C05476=1182.261,381.799,-80.874,-176.029,8.760,148.599
C05477=1182.257,382.046,-80.909,-176.028,8.763,148.599
C05478=1182.253,382.294,-80.944,-176.027,8.766,148.600
C05479=1182.249,382.541,-80.980,-176.026,8.769,148.600
C05480=1182.245,382.789,-81.014,-176.026,8.772,148.601
C05481=1182.241,383.036,-81.050,-176.024,8.776,148.601
C05482=1182.238,383.284,-81.085,-176.023,8.779,148.602
C05483=1182.233,383.531,-81.120,-176.023,8.783,148.603
C05484=1182.229,383.779,-81.155,-176.022,8.786,148.603
C05485=1182.225,384.027,-81.190,-176.021,8.789,148.604
C05486=1182.221,384.274,-81.225,-176.020,8.792,148.605
C05487=1182.217,384.521,-81.261,-176.020,8.795,148.605
C05488=1182.214,384.769,-81.296,-176.019,8.798,148.606
C05489=1182.209,385.016,-81.331,-176.019,8.800,148.606
C05490=1182.206,385.264,-81.366,-176.018,8.804,148.607
C05491=1182.202,385.512,-81.401,-176.017,8.807,148.608
C05492=1182.197,385.759,-81.436,-176.017,8.810,148.608
C05493=1182.194,386.006,-81.472,-176.016,8.813,148.609
C05494=1182.190,386.254,-81.507,-176.015,8.816,148.610
C05495=1182.185,386.501,-81.542,-176.015,8.819,148.610
C05496=1182.182,386.748,-81.577,-176.014,8.822,148.611
C05497=1182.178,386.996,-81.613,-176.013,8.825,148.611
C05498=1182.174,387.243,-81.649,-176.013,8.828,148.612
C05499=1182.170,387.491,-81.683,-176.012,8.831,148.613
C05500=1182.165,387.739,-81.719,-176.012,8.834,148.613
C05501=1182.162,387.986,-81.755,-176.012,8.837,148.614
C05502=1182.158,388.233,-81.790,-176.011,8.840,148.615
C05503=1182.154,388.481,-81.825,-176.010,8.843,148.615
C05504=1182.150,388.729,-81.860,-176.010,8.846,148.616
C05505=1182.146,388.976,-81.896,-176.009,8.849,148.616
C05506=1182.142,389.223,-81.931,-176.009,8.852,148.617
C05507=1182.138,389.470,-81.967,-176.009,8.854,148.618
C05508=1182.134,389.719,-82.001,-176.008,8.858,148.618
C05509=1182.130,389.965,-82.037,-176.008,8.860,148.619
C05510=1182.126,390.213,-82.072,-176.007,8.863,148.620
C05511=1182.122,390.461,-82.108,-176.007,8.866,148.620
C05512=1182.118,390.708,-82.144,-176.007,8.869,148.621
C05513=1182.114,390.955,-82.179,-176.007,8.871,148.622
C05514=1182.110,391.203,-82.214,-176.006,8.875,148.622
C05515=1182.106,391.451,-82.249,-176.006,8.877,148.623
C05516=1182.102,391.734,-82.290,-176.005,8.880,148.624
C05517=1182.098,392.019,-82.331,-176.005,8.884,148.624
C05518=1182.093,392.302,-82.372,-176.005,8.887,148.625
C05519=1182.088,392.586,-82.412,-176.004,8.890,148.626
C05520=1182.084,392.834,-82.448,-176.004,8.893,148.626
C05521=1182.081,393.081,-82.483,-176.004,8.895,148.627
C05522=1182.077,393.329,-82.519,-176.003,8.898,148.628
C05523=1182.072,393.576,-82.554,-176.003,8.901,148.628
C05524=1182.068,393.823,-82.590,-176.003,8.903,148.629
C05525=1182.065,394.071,-82.626,-176.003,8.907,148.630
C05526=1182.061,394.318,-82.661,-176.003,8.909,148.630
C05527=1182.057,394.565,-82.696,-176.003,8.911,148.631
C05528=1182.053,394.813,-82.732,-176.002,8.914,148.632
C05529=1182.049,395.061,-82.768,-176.002,8.917,148.632
C05530=1182.045,395.309,-82.803,-176.002,8.919,148.633
C05531=1182.041,395.556,-82.838,-176.002,8.922,148.633
C05532=1182.037,395.803,-82.874,-176.001,8.925,148.634
C05533=1182.033,396.051,-82.909,-176.001,8.928,148.635
C05534=1182.029,396.298,-82.945,-176.001,8.930,148.635
C05535=1182.025,396.546,-82.981,-176.001,8.932,148.636
C05536=1182.021,396.793,-83.016,-176.001,8.935,148.637
C05537=1182.017,397.040,-83.051,-176.001,8.937,148.637
C05538=1182.014,397.288,-83.087,-176.000,8.940,148.638
C05539=1182.009,397.535,-83.123,-176.001,8.943,148.639
C05540=1182.005,397.783,-83.159,-176.000,8.945,148.639
C05541=1182.001,398.030,-83.194,-176.000,8.948,148.640
C05542=1181.998,398.277,-83.229,-176.000,8.950,148.640
C05543=1181.993,398.525,-83.266,-176.000,8.953,148.641
C05544=1181.989,398.773,-83.301,-176.000,8.955,148.642
C05545=1181.985,399.019,-83.336,-176.000,8.957,148.642
C05546=1181.982,399.267,-83.372,-176.000,8.960,148.643
C05547=1181.977,399.515,-83.408,-176.000,8.962,148.644
C05548=1181.974,399.762,-83.444,-176.000,8.964,148.644
C05549=1181.970,400.010,-83.479,-176.000,8.967,148.645
C05550=1181.966,400.257,-83.515,-176.000,8.969,148.645
C05551=1181.961,400.504,-83.551,-176.000,8.972,148.646
C05552=1181.958,400.751,-83.587,-176.000,8.974,148.647
C05553=1181.954,400.999,-83.622,-176.000,8.977,148.647
C05554=1181.950,401.246,-83.658,-176.000,8.979,148.648
C05555=1181.946,401.494,-83.694,-176.000,8.982,148.649
C05556=1181.942,401.741,-83.729,-176.000,8.984,148.649
C05557=1181.938,401.988,-83.765,-176.000,8.986,148.650
C05558=1181.935,402.236,-83.800,-175.999,8.989,148.650
C05559=1181.930,402.484,-83.836,-176.000,8.991,148.651
C05560=1181.926,402.731,-83.872,-175.999,8.993,148.652
C05561=1181.922,402.978,-83.907,-175.999,8.996,148.652
C05562=1181.918,403.226,-83.943,-176.000,8.997,148.653
C05563=1181.914,403.473,-83.979,-176.000,9.000,148.653
C05564=1181.911,403.720,-84.015,-176.000,9.002,148.654
C05565=1181.907,403.968,-84.051,-176.000,9.005,148.654
C05566=1181.903,404.215,-84.087,-176.000,9.007,148.655
C05567=1181.898,404.462,-84.122,-175.999,9.009,148.656
C05568=1181.895,404.710,-84.157,-176.000,9.011,148.656
C05569=1181.890,404.957,-84.194,-176.000,9.013,148.657
C05570=1181.887,405.205,-84.229,-176.000,9.016,148.657
C05571=1181.883,405.452,-84.265,-176.000,9.018,148.658
C05572=1181.879,405.700,-84.302,-176.000,9.020,148.659
C05573=1181.875,405.947,-84.337,-176.000,9.022,148.659
C05574=1181.871,406.194,-84.372,-176.000,9.024,148.660
C05575=1181.867,406.441,-84.408,-176.000,9.027,148.660
C05576=1181.863,406.689,-84.444,-176.000,9.029,148.661
C05577=1181.859,406.937,-84.480,-176.000,9.031,148.662
C05578=1181.856,407.184,-84.516,-176.000,9.033,148.662
C05579=1181.852,407.431,-84.552,-176.000,9.036,148.663
C05580=1181.847,407.678,-84.587,-176.000,9.038,148.663
C05581=1181.844,407.926,-84.623,-176.000,9.039,148.664
C05582=1181.839,408.174,-84.659,-176.000,9.042,148.664
C05583=1181.836,408.420,-84.695,-176.000,9.044,148.665
C05584=1181.832,408.668,-84.731,-176.000,9.046,148.665
C05585=1181.828,408.916,-84.767,-176.001,9.048,148.666
C05586=1181.824,409.163,-84.802,-176.000,9.050,148.667
C05587=1181.820,409.410,-84.837,-176.001,9.052,148.667
C05588=1181.816,409.657,-84.874,-176.001,9.054,148.668
C05589=1181.812,409.905,-84.910,-176.000,9.057,148.668
C05590=1181.808,410.152,-84.945,-176.001,9.058,148.669
C05591=1181.804,410.400,-84.982,-176.001,9.061,148.670
C05592=1181.800,410.648,-85.017,-176.001,9.063,148.670
C05593=1181.797,410.894,-85.053,-176.001,9.064,148.671
C05594=1181.793,411.142,-85.090,-176.001,9.067,148.671
C05595=1181.788,411.389,-85.125,-176.001,9.068,148.672
C05596=1181.784,411.637,-85.161,-176.001,9.071,148.672
C05597=1181.781,411.884,-85.197,-176.001,9.073,148.673
C05598=1181.777,412.131,-85.233,-176.001,9.074,148.673
C05599=1181.773,412.379,-85.269,-176.001,9.077,148.674
C05600=1181.769,412.627,-85.304,-176.002,9.078,148.674
C05601=1181.765,412.874,-85.340,-176.001,9.081,148.675
C05602=1181.761,413.121,-85.377,-176.002,9.082,148.675
C05603=1181.757,413.368,-85.412,-176.001,9.084,148.676
C05604=1181.752,413.616,-85.448,-176.002,9.087,148.677
C05605=1181.749,413.863,-85.484,-176.002,9.088,148.677
C05606=1181.745,414.110,-85.520,-176.002,9.091,148.678
C05607=1181.741,414.358,-85.556,-176.002,9.092,148.678
C05608=1181.737,414.606,-85.592,-176.002,9.094,148.679
C05609=1181.734,414.852,-85.628,-176.002,9.096,148.679
C05610=1181.730,415.100,-85.664,-176.002,9.098,148.680
C05611=1181.726,415.348,-85.700,-176.002,9.100,148.680
C05612=1181.722,415.571,-85.732,-176.002,9.102,148.681
C05613=1181.718,415.796,-85.765,-176.002,9.103,148.681
C05614=1181.716,416.020,-85.797,-176.003,9.105,148.682
C05615=1181.714,416.244,-85.830,-176.002,9.107,148.682
C05616=1181.714,416.467,-85.862,-176.002,9.108,148.682
C05617=1181.715,416.691,-85.894,-176.003,9.110,148.683
C05618=1181.716,416.915,-85.927,-176.002,9.112,148.683
C05619=1181.719,417.138,-85.958,-176.002,9.113,148.684
C05620=1181.298,417.140,-86.000,-176.006,9.124,148.687
C05621=1181.295,416.914,-85.968,-176.005,9.123,148.687
C05622=1181.293,416.689,-85.936,-176.006,9.120,148.687
C05623=1181.293,416.464,-85.903,-176.006,9.119,148.686
C05624=1181.294,416.238,-85.871,-176.005,9.118,148.686
C05625=1181.295,416.013,-85.838,-176.006,9.115,148.685
C05626=1181.297,415.788,-85.806,-176.005,9.114,148.685
C05627=1181.301,415.563,-85.773,-176.005,9.113,148.684
C05628=1181.305,415.336,-85.740,-176.005,9.110,148.684
C05629=1181.308,415.089,-85.704,-176.005,9.109,148.683
C05630=1181.312,414.841,-85.668,-176.005,9.107,148.683
C05631=1181.316,414.594,-85.632,-176.005,9.105,148.682
C05632=1181.320,414.347,-85.596,-176.005,9.103,148.682
C05633=1181.324,414.100,-85.560,-176.005,9.101,148.681
C05634=1181.328,413.852,-85.525,-176.005,9.099,148.681
C05635=1181.332,413.605,-85.489,-176.005,9.098,148.680
C05636=1181.336,413.357,-85.452,-176.005,9.095,148.680
C05637=1181.339,413.110,-85.417,-176.005,9.094,148.679
C05638=1181.344,412.862,-85.381,-176.004,9.091,148.679
C05639=1181.347,412.615,-85.345,-176.005,9.089,148.678
C05640=1181.351,412.368,-85.309,-176.004,9.088,148.678
C05641=1181.356,412.121,-85.273,-176.005,9.085,148.677
C05642=1181.359,411.873,-85.238,-176.004,9.084,148.676
C05643=1181.364,411.625,-85.201,-176.004,9.081,148.676
C05644=1181.367,411.378,-85.165,-176.004,9.080,148.675
C05645=1181.371,411.131,-85.130,-176.004,9.078,148.675
C05646=1181.375,410.883,-85.093,-176.004,9.075,148.674
C05647=1181.379,410.636,-85.058,-176.004,9.074,148.674
C05648=1181.382,410.389,-85.022,-176.004,9.071,148.673
C05649=1181.387,410.142,-84.986,-176.004,9.069,148.672
C05650=1181.391,409.894,-84.950,-176.003,9.067,148.672
C05651=1181.395,409.647,-84.915,-176.004,9.065,148.671
C05652=1181.399,409.399,-84.878,-176.003,9.064,148.671
C05653=1181.402,409.152,-84.842,-176.003,9.061,148.670
C05654=1181.406,408.904,-84.807,-176.004,9.059,148.670
C05655=1181.410,408.657,-84.771,-176.003,9.057,148.669
C05656=1181.415,408.410,-84.735,-176.003,9.055,148.669
C05657=1181.418,408.163,-84.699,-176.003,9.053,148.668
C05658=1181.422,407.915,-84.663,-176.003,9.051,148.668
C05659=1181.426,407.668,-84.628,-176.003,9.049,148.667
C05660=1181.430,407.420,-84.592,-176.003,9.046,148.666
C05661=1181.434,407.172,-84.556,-176.003,9.044,148.666
C05662=1181.438,406.925,-84.520,-176.003,9.042,148.665
C05663=1181.442,406.679,-84.484,-176.003,9.040,148.665
C05664=1181.446,406.431,-84.448,-176.003,9.037,148.664
C05665=1181.450,406.183,-84.413,-176.002,9.036,148.664
C05666=1181.454,405.936,-84.377,-176.002,9.033,148.663
C05667=1181.458,405.688,-84.341,-176.003,9.031,148.662
C05668=1181.462,405.441,-84.305,-176.003,9.029,148.662
C05669=1181.465,405.194,-84.269,-176.003,9.026,148.661
C05670=1181.470,404.947,-84.233,-176.002,9.025,148.661
C05671=1181.474,404.699,-84.198,-176.002,9.022,148.660
C05672=1181.477,404.452,-84.162,-176.002,9.020,148.659
C05673=1181.482,404.204,-84.126,-176.002,9.017,148.659
C05674=1181.485,403.956,-84.091,-176.003,9.015,148.658
C05675=1181.489,403.709,-84.055,-176.002,9.014,148.658
C05676=1181.493,403.463,-84.019,-176.002,9.011,148.657
C05677=1181.497,403.215,-83.983,-176.002,9.009,148.656
C05678=1181.501,402.967,-83.948,-176.002,9.006,148.656
C05679=1181.505,402.720,-83.912,-176.002,9.004,148.655
C05680=1181.509,402.472,-83.876,-176.002,9.002,148.654
C05681=1181.513,402.224,-83.840,-176.003,8.999,148.654
C05682=1181.517,401.978,-83.805,-176.002,8.997,148.653
C05683=1181.521,401.730,-83.770,-176.002,8.995,148.653
C05684=1181.525,401.482,-83.733,-176.002,8.993,148.652
C05685=1181.529,401.235,-83.698,-176.002,8.990,148.651
C05686=1181.532,400.988,-83.662,-176.002,8.988,148.651
C05687=1181.537,400.740,-83.625,-176.002,8.986,148.650
C05688=1181.541,400.493,-83.590,-176.002,8.983,148.650
C05689=1181.544,400.246,-83.555,-176.002,8.981,148.649
C05690=1181.548,399.998,-83.519,-176.002,8.978,148.648
C05691=1181.553,399.751,-83.483,-176.002,8.976,148.648
C05692=1181.556,399.503,-83.447,-176.002,8.973,148.647
C05693=1181.560,399.256,-83.412,-176.002,8.971,148.647
C05694=1181.564,399.009,-83.377,-176.002,8.969,148.646
C05695=1181.569,398.761,-83.341,-176.003,8.966,148.645
C05696=1181.572,398.513,-83.305,-176.002,8.964,148.645
C05697=1181.576,398.266,-83.270,-176.003,8.961,148.644
C05698=1181.580,398.019,-83.234,-176.002,8.959,148.643
C05699=1181.585,397.771,-83.198,-176.003,8.956,148.643
C05700=1181.588,397.524,-83.163,-176.003,8.953,148.642
C05701=1181.592,397.276,-83.127,-176.003,8.951,148.642
C05702=1181.595,397.029,-83.092,-176.003,8.948,148.641
C05703=1181.600,396.782,-83.056,-176.003,8.946,148.640
C05704=1181.604,396.534,-83.020,-176.003,8.944,148.640
C05705=1181.608,396.287,-82.985,-176.004,8.941,148.639
C05706=1181.611,396.039,-82.949,-176.004,8.938,148.638
C05707=1181.616,395.792,-82.914,-176.004,8.936,148.638
C05708=1181.620,395.545,-82.878,-176.004,8.933,148.637
C05709=1181.624,395.297,-82.842,-176.004,8.930,148.636
C05710=1181.627,395.050,-82.807,-176.004,8.928,148.636
C05711=1181.631,394.802,-82.771,-176.005,8.925,148.635
C05712=1181.635,394.555,-82.736,-176.005,8.923,148.634
C05713=1181.640,394.308,-82.700,-176.005,8.920,148.634
C05714=1181.643,394.060,-82.664,-176.005,8.917,148.633
C05715=1181.647,393.813,-82.629,-176.005,8.914,148.632
C05716=1181.651,393.566,-82.594,-176.005,8.912,148.632
C05717=1181.655,393.318,-82.558,-176.006,8.909,148.631
C05718=1181.659,393.071,-82.522,-176.006,8.906,148.631
C05719=1181.663,392.822,-82.487,-176.006,8.904,148.630
C05720=1181.667,392.575,-82.451,-176.007,8.901,148.629
C05721=1181.672,392.291,-82.411,-176.007,8.898,148.629
C05722=1181.676,392.007,-82.371,-176.007,8.895,148.628
C05723=1181.680,391.723,-82.329,-176.007,8.891,148.627
C05724=1181.686,391.439,-82.289,-176.008,8.888,148.626
C05725=1181.689,391.191,-82.253,-176.008,8.886,148.626
C05726=1181.693,390.944,-82.218,-176.009,8.883,148.625
C05727=1181.697,390.697,-82.183,-176.009,8.880,148.624
C05728=1181.701,390.450,-82.147,-176.009,8.877,148.624
C05729=1181.704,390.202,-82.111,-176.009,8.874,148.623
C05730=1181.708,389.955,-82.076,-176.010,8.871,148.623
C05731=1181.713,389.707,-82.041,-176.010,8.869,148.622
C05732=1181.717,389.459,-82.005,-176.011,8.866,148.621
C05733=1181.721,389.212,-81.970,-176.012,8.863,148.621
C05734=1181.725,388.965,-81.935,-176.011,8.860,148.620
C05735=1181.729,388.718,-81.899,-176.012,8.857,148.619
C05736=1181.733,388.470,-81.864,-176.013,8.854,148.619
C05737=1181.736,388.222,-81.829,-176.013,8.851,148.618
C05738=1181.741,387.975,-81.793,-176.014,8.848,148.617
C05739=1181.744,387.728,-81.758,-176.014,8.845,148.617
C05740=1181.748,387.480,-81.722,-176.014,8.842,148.616
C05741=1181.752,387.233,-81.688,-176.015,8.839,148.616
C05742=1181.757,386.985,-81.652,-176.016,8.836,148.615
C05743=1181.761,386.737,-81.616,-176.016,8.833,148.614
C05744=1181.764,386.490,-81.581,-176.017,8.830,148.614
C05745=1181.769,386.243,-81.546,-176.017,8.827,148.613
C05746=1181.772,385.995,-81.511,-176.018,8.824,148.612
C05747=1181.776,385.748,-81.475,-176.019,8.821,148.612
C05748=1181.780,385.501,-81.440,-176.019,8.818,148.611
C05749=1181.784,385.253,-81.405,-176.020,8.815,148.610
C05750=1181.788,385.005,-81.370,-176.021,8.811,148.610
C05751=1181.792,384.758,-81.334,-176.021,8.808,148.609
C05752=1181.796,384.510,-81.300,-176.022,8.805,148.609
C05753=1181.800,384.263,-81.264,-176.023,8.802,148.608
C05754=1181.804,384.016,-81.229,-176.024,8.799,148.607
C05755=1181.808,383.768,-81.194,-176.024,8.796,148.607
C05756=1181.812,383.520,-81.158,-176.025,8.793,148.606
C05757=1181.816,383.274,-81.123,-176.026,8.790,148.606
C05758=1181.820,383.025,-81.088,-176.027,8.786,148.605
C05759=1181.824,382.778,-81.053,-176.028,8.783,148.604
C05760=1181.828,382.531,-81.018,-176.028,8.780,148.604
C05761=1181.832,382.283,-80.983,-176.029,8.777,148.603
C05762=1181.836,382.035,-80.947,-176.030,8.774,148.603
C05763=1181.840,381.788,-80.913,-176.031,8.771,148.602
C05764=1181.844,381.541,-80.877,-176.031,8.768,148.601
C05765=1181.848,381.292,-80.842,-176.033,8.764,148.601
C05766=1181.852,381.046,-80.807,-176.033,8.761,148.600
C05767=1181.856,380.798,-80.772,-176.035,8.758,148.600
C05768=1181.860,380.551,-80.737,-176.036,8.755,148.599
C05769=1181.864,380.303,-80.702,-176.036,8.752,148.599
C05770=1181.868,380.055,-80.667,-176.038,8.748,148.598
C05771=1181.872,379.808,-80.632,-176.039,8.745,148.597
C05772=1181.875,379.560,-80.597,-176.039,8.741,148.597
C05773=1181.879,379.313,-80.562,-176.040,8.738,148.596
C05774=1181.884,379.066,-80.527,-176.042,8.734,148.595
C05775=1181.887,378.818,-80.492,-176.042,8.731,148.595
C05776=1181.892,378.571,-80.457,-176.043,8.728,148.594
C05777=1181.895,378.323,-80.422,-176.045,8.725,148.594
C05778=1181.899,378.075,-80.387,-176.046,8.722,148.593
C05779=1181.904,377.828,-80.352,-176.047,8.718,148.593
C05780=1181.908,377.580,-80.317,-176.048,8.715,148.592
C05781=1181.912,377.333,-80.283,-176.049,8.711,148.592
C05782=1181.915,377.085,-80.248,-176.051,8.708,148.591
C05783=1181.920,376.838,-80.213,-176.052,8.705,148.590
C05784=1181.923,376.591,-80.178,-176.053,8.701,148.590
C05785=1181.927,376.342,-80.143,-176.054,8.698,148.589
C05786=1181.932,376.095,-80.108,-176.056,8.694,148.589
C05787=1181.936,375.848,-80.073,-176.056,8.691,148.588
C05788=1181.939,375.600,-80.039,-176.058,8.688,148.588
C05789=1181.943,375.353,-80.003,-176.059,8.684,148.587
C05790=1181.948,375.106,-79.969,-176.060,8.680,148.587
C05791=1181.952,374.857,-79.934,-176.062,8.678,148.586
C05792=1181.956,374.611,-79.899,-176.063,8.674,148.586
C05793=1181.959,374.363,-79.865,-176.064,8.671,148.585
C05794=1181.963,374.115,-79.830,-176.066,8.667,148.585
C05795=1181.968,373.867,-79.795,-176.067,8.664,148.584
C05796=1181.971,373.620,-79.760,-176.068,8.660,148.584
C05797=1181.975,373.373,-79.726,-176.070,8.657,148.583
C05798=1181.979,373.125,-79.691,-176.071,8.653,148.583
C05799=1181.984,372.877,-79.657,-176.073,8.650,148.582
C05800=1181.987,372.630,-79.621,-176.074,8.647,148.582
C05801=1181.991,372.382,-79.587,-176.075,8.643,148.581
C05802=1181.995,372.134,-79.552,-176.077,8.639,148.580
C05803=1182.000,371.887,-79.518,-176.078,8.636,148.580
C05804=1182.003,371.639,-79.482,-176.080,8.633,148.580
C05805=1182.007,371.392,-79.448,-176.081,8.629,148.579
C05806=1182.011,371.144,-79.414,-176.082,8.626,148.579
C05807=1182.016,370.897,-79.379,-176.084,8.622,148.578
C05808=1182.019,370.649,-79.345,-176.086,8.619,148.578
C05809=1182.024,370.402,-79.310,-176.087,8.616,148.577
C05810=1182.028,370.153,-79.276,-176.089,8.612,148.577
C05811=1182.031,369.907,-79.241,-176.090,8.608,148.576
C05812=1182.035,369.659,-79.206,-176.092,8.605,148.576
C05813=1182.040,369.411,-79.172,-176.093,8.602,148.575
C05814=1182.043,369.164,-79.138,-176.095,8.598,148.575
C05815=1182.047,368.916,-79.103,-176.097,8.595,148.574
C05816=1182.052,368.669,-79.069,-176.098,8.591,148.574
C05817=1182.055,368.421,-79.034,-176.100,8.587,148.573
C05818=1182.060,368.174,-79.000,-176.101,8.584,148.573
C05819=1182.064,367.925,-78.965,-176.103,8.581,148.573
C05820=1182.068,367.678,-78.931,-176.105,8.577,148.572
C05821=1182.072,367.430,-78.896,-176.107,8.573,148.572
C05822=1182.075,367.183,-78.862,-176.109,8.570,148.571
C05823=1182.080,366.936,-78.828,-176.110,8.566,148.571
C05824=1182.084,366.688,-78.793,-176.112,8.563,148.570
C05825=1182.088,366.406,-78.754,-176.114,8.559,148.570
C05826=1182.092,366.125,-78.715,-176.116,8.555,148.570
C05827=1182.097,365.843,-78.676,-176.118,8.551,148.569
C05828=1182.102,365.561,-78.638,-176.120,8.547,148.568
C05829=1182.106,365.314,-78.603,-176.122,8.544,148.568
C05830=1182.110,365.067,-78.570,-176.124,8.540,148.568
C05831=1182.114,364.819,-78.535,-176.125,8.536,148.567
C05832=1182.118,364.572,-78.501,-176.127,8.533,148.567
C05833=1182.122,364.323,-78.466,-176.129,8.530,148.567
C05834=1182.126,364.076,-78.432,-176.130,8.526,148.566
C05835=1182.130,363.828,-78.398,-176.132,8.523,148.566
C05836=1182.134,363.580,-78.364,-176.134,8.519,148.565
C05837=1182.138,363.333,-78.330,-176.136,8.516,148.565
C05838=1182.142,363.086,-78.296,-176.138,8.512,148.565
C05839=1182.146,362.838,-78.261,-176.140,8.509,148.564
C05840=1182.150,362.590,-78.228,-176.142,8.505,148.564
C05841=1182.155,362.343,-78.193,-176.144,8.502,148.563
C05842=1182.158,362.095,-78.159,-176.146,8.498,148.563
C05843=1182.162,361.848,-78.125,-176.148,8.494,148.563
C05844=1182.167,361.600,-78.091,-176.150,8.491,148.562
C05845=1182.170,361.352,-78.057,-176.152,8.487,148.562
C05846=1182.174,361.104,-78.023,-176.153,8.484,148.562
C05847=1182.179,360.857,-77.990,-176.156,8.480,148.561
C05848=1182.182,360.609,-77.955,-176.158,8.477,148.561
C05849=1182.186,360.362,-77.921,-176.160,8.474,148.561
C05850=1182.191,360.114,-77.888,-176.162,8.470,148.560
C05851=1182.195,359.866,-77.853,-176.164,8.467,148.560
C05852=1182.198,359.619,-77.819,-176.166,8.463,148.560
C05853=1182.202,359.371,-77.786,-176.168,8.459,148.559
C05854=1182.207,359.123,-77.751,-176.170,8.456,148.559
C05855=1182.211,358.875,-77.718,-176.172,8.452,148.558
C05856=1182.214,358.628,-77.684,-176.174,8.449,148.558
C05857=1182.219,358.380,-77.650,-176.176,8.446,148.558
C05858=1182.223,358.132,-77.616,-176.178,8.442,148.558
C05859=1182.226,357.885,-77.582,-176.180,8.439,148.557
C05860=1182.231,357.637,-77.548,-176.182,8.435,148.557
C05861=1182.235,357.390,-77.515,-176.184,8.432,148.557
C05862=1182.239,357.141,-77.481,-176.186,8.428,148.556
C05863=1182.242,356.894,-77.447,-176.188,8.425,148.556
C05864=1182.247,356.646,-77.413,-176.191,8.422,148.556
C05865=1182.251,356.399,-77.380,-176.192,8.418,148.555
C05866=1182.255,356.151,-77.346,-176.195,8.415,148.555
C05867=1182.259,355.903,-77.313,-176.197,8.411,148.555
C05868=1182.263,355.655,-77.278,-176.199,8.407,148.554
C05869=1182.268,355.408,-77.245,-176.202,8.404,148.554
C05870=1182.271,355.161,-77.211,-176.204,8.400,148.554
C05871=1182.275,354.913,-77.178,-176.206,8.397,148.554
C05872=1182.279,354.664,-77.145,-176.208,8.393,148.553
C05873=1182.284,354.417,-77.110,-176.210,8.390,148.553
C05874=1182.288,354.169,-77.077,-176.212,8.386,148.553
C05875=1182.292,353.922,-77.044,-176.214,8.383,148.553
C05876=1182.296,353.675,-77.010,-176.217,8.380,148.552
C05877=1182.300,353.427,-76.977,-176.219,8.377,148.552
C05878=1182.303,353.178,-76.943,-176.221,8.373,148.552
C05879=1182.308,352.931,-76.909,-176.223,8.370,148.551
C05880=1182.312,352.683,-76.876,-176.225,8.366,148.551
C05881=1182.316,352.435,-76.843,-176.227,8.363,148.551
C05882=1182.320,352.188,-76.809,-176.229,8.359,148.551
C05883=1182.324,351.941,-76.776,-176.231,8.356,148.550
C05884=1182.328,351.693,-76.742,-176.234,8.353,148.550
C05885=1182.332,351.444,-76.709,-176.236,8.349,148.550
C05886=1182.336,351.197,-76.676,-176.238,8.346,148.550
C05887=1182.341,350.949,-76.642,-176.240,8.343,148.549
C05888=1182.345,350.701,-76.609,-176.242,8.339,148.549
C05889=1182.349,350.454,-76.575,-176.245,8.336,148.549
C05890=1182.353,350.206,-76.542,-176.247,8.333,148.549
C05891=1182.357,349.958,-76.509,-176.249,8.329,148.548
C05892=1182.361,349.711,-76.475,-176.251,8.326,148.548
C05893=1182.365,349.463,-76.442,-176.254,8.323,148.548
C05894=1182.369,349.215,-76.409,-176.256,8.319,148.548
C05895=1182.373,348.967,-76.376,-176.258,8.316,148.547
C05896=1182.377,348.719,-76.342,-176.260,8.312,148.547
C05897=1182.381,348.471,-76.309,-176.262,8.309,148.547
C05898=1182.385,348.224,-76.276,-176.265,8.305,148.547
C05899=1182.390,347.976,-76.243,-176.267,8.302,148.546
C05900=1182.394,347.728,-76.210,-176.270,8.298,148.546
C05901=1182.398,347.480,-76.177,-176.272,8.295,148.546
C05902=1182.402,347.233,-76.144,-176.274,8.292,148.546
C05903=1182.406,346.985,-76.110,-176.276,8.288,148.545
C05904=1182.410,346.737,-76.077,-176.279,8.285,148.545
C05905=1182.414,346.489,-76.044,-176.281,8.282,148.545
C05906=1182.419,346.242,-76.011,-176.283,8.278,148.545
C05907=1182.423,345.994,-75.978,-176.285,8.275,148.545
C05908=1182.427,345.746,-75.945,-176.288,8.272,148.544
C05909=1182.430,345.499,-75.912,-176.290,8.268,148.544
C05910=1182.434,345.251,-75.879,-176.292,8.265,148.544
C05911=1182.439,345.003,-75.846,-176.294,8.262,148.544
C05912=1182.443,344.755,-75.813,-176.297,8.258,148.544
C05913=1182.447,344.507,-75.780,-176.299,8.255,148.543
C05914=1182.451,344.260,-75.747,-176.301,8.252,148.543
C05915=1182.455,344.012,-75.714,-176.303,8.249,148.543
C05916=1182.460,343.764,-75.681,-176.306,8.245,148.543
C05917=1182.463,343.516,-75.649,-176.308,8.242,148.542
C05918=1182.467,343.268,-75.616,-176.310,8.239,148.542
C05919=1182.472,343.021,-75.583,-176.312,8.235,148.542
C05920=1182.476,342.772,-75.550,-176.315,8.232,148.542
C05921=1182.480,342.525,-75.517,-176.317,8.229,148.542
C05922=1182.484,342.277,-75.484,-176.320,8.226,148.542
C05923=1182.488,342.029,-75.451,-176.322,8.222,148.541
C05924=1182.493,341.782,-75.419,-176.324,8.219,148.541
C05925=1182.497,341.534,-75.386,-176.326,8.216,148.541
C05926=1182.501,341.286,-75.353,-176.329,8.212,148.541
C05927=1182.505,341.038,-75.320,-176.331,8.209,148.540
C05928=1182.509,340.791,-75.288,-176.333,8.206,148.540
C05929=1182.514,340.512,-75.251,-176.336,8.203,148.540
C05930=1182.518,340.232,-75.214,-176.339,8.199,148.540
C05931=1182.523,339.953,-75.178,-176.341,8.195,148.540
C05932=1182.528,339.674,-75.141,-176.344,8.191,148.540
C05933=1182.532,339.427,-75.108,-176.346,8.188,148.539
C05934=1182.536,339.179,-75.076,-176.348,8.185,148.539
C05935=1182.540,338.931,-75.043,-176.351,8.181,148.539
C05936=1182.544,338.683,-75.010,-176.353,8.178,148.539
C05937=1182.548,338.435,-74.978,-176.356,8.175,148.539
C05938=1182.553,338.187,-74.945,-176.358,8.172,148.538
C05939=1182.557,337.940,-74.912,-176.360,8.168,148.538
C05940=1182.561,337.692,-74.880,-176.363,8.165,148.538
C05941=1182.565,337.444,-74.847,-176.365,8.162,148.538
C05942=1182.568,337.196,-74.815,-176.367,8.159,148.538
C05943=1182.573,336.948,-74.782,-176.369,8.156,148.538
C05944=1182.578,336.701,-74.750,-176.372,8.153,148.538
C05945=1182.581,336.453,-74.718,-176.374,8.150,148.537
C05946=1182.585,336.205,-74.685,-176.376,8.146,148.537
C05947=1182.589,335.957,-74.653,-176.379,8.143,148.537
C05948=1182.593,335.709,-74.620,-176.381,8.140,148.537
C05949=1182.598,335.461,-74.588,-176.384,8.137,148.537
C05950=1182.602,335.213,-74.556,-176.386,8.134,148.537
C05951=1182.606,334.966,-74.523,-176.388,8.130,148.536
C05952=1182.610,334.718,-74.491,-176.391,8.127,148.536
C05953=1182.614,334.469,-74.459,-176.393,8.124,148.536
C05954=1182.618,334.222,-74.426,-176.395,8.121,148.536
C05955=1182.623,333.974,-74.394,-176.398,8.118,148.536
C05956=1182.626,333.726,-74.362,-176.400,8.114,148.536
C05957=1182.631,333.478,-74.330,-176.403,8.111,148.536
C05958=1182.634,333.230,-74.297,-176.405,8.108,148.536
C05959=1182.639,332.983,-74.265,-176.407,8.105,148.535
C05960=1182.643,332.735,-74.233,-176.410,8.101,148.535
C05961=1182.648,332.486,-74.201,-176.412,8.098,148.535
C05962=1182.651,332.238,-74.169,-176.415,8.095,148.535
C05963=1182.656,331.991,-74.136,-176.417,8.092,148.535
C05964=1182.660,331.743,-74.105,-176.420,8.089,148.535
C05965=1182.664,331.495,-74.072,-176.422,8.085,148.534
C05966=1182.668,331.247,-74.040,-176.424,8.082,148.534
C05967=1182.673,330.999,-74.008,-176.427,8.079,148.534
C05968=1182.677,330.751,-73.976,-176.429,8.076,148.534
C05969=1182.680,330.503,-73.944,-176.431,8.072,148.534
C05970=1182.685,330.255,-73.912,-176.434,8.069,148.534
C05971=1182.689,330.008,-73.880,-176.436,8.066,148.534
C05972=1182.693,329.760,-73.847,-176.439,8.063,148.534
C05973=1182.697,329.512,-73.816,-176.441,8.061,148.533
C05974=1182.701,329.264,-73.784,-176.443,8.057,148.533
C05975=1182.706,329.016,-73.752,-176.446,8.054,148.533
C05976=1182.709,328.768,-73.720,-176.448,8.051,148.533
C05977=1182.714,328.521,-73.688,-176.451,8.048,148.533
C05978=1182.718,328.272,-73.656,-176.453,8.045,148.533
C05979=1182.722,328.024,-73.624,-176.456,8.042,148.533
C05980=1182.726,327.777,-73.593,-176.458,8.038,148.533
C05981=1182.731,327.528,-73.561,-176.460,8.035,148.532
C05982=1182.735,327.281,-73.529,-176.463,8.032,148.532
C05983=1182.739,327.032,-73.498,-176.465,8.029,148.532
C05984=1182.743,326.784,-73.466,-176.468,8.026,148.532
C05985=1182.748,326.537,-73.434,-176.470,8.022,148.532
C05986=1182.751,326.289,-73.402,-176.473,8.019,148.532
C05987=1182.755,326.041,-73.370,-176.475,8.016,148.532
C05988=1182.760,325.793,-73.338,-176.478,8.013,148.532
C05989=1182.764,325.544,-73.307,-176.480,8.010,148.532
C05990=1182.768,325.297,-73.275,-176.483,8.007,148.532
C05991=1182.772,325.049,-73.243,-176.485,8.003,148.531
C05992=1182.776,324.801,-73.212,-176.487,8.001,148.531
C05993=1182.781,324.553,-73.179,-176.490,7.998,148.531
C05994=1182.785,324.305,-73.148,-176.492,7.995,148.531
C05995=1182.789,324.057,-73.117,-176.494,7.992,148.531
C05996=1182.793,323.809,-73.085,-176.497,7.988,148.531
C05997=1182.797,323.561,-73.053,-176.499,7.985,148.531
C05998=1182.801,323.313,-73.022,-176.502,7.982,148.531
C05999=1182.806,323.065,-72.990,-176.504,7.979,148.531
C06000=1182.810,322.818,-72.958,-176.507,7.976,148.531
C06001=1182.814,322.569,-72.927,-176.509,7.973,148.530
C06002=1182.818,322.322,-72.896,-176.512,7.970,148.530
C06003=1182.822,322.074,-72.864,-176.514,7.966,148.530
C06004=1182.826,321.825,-72.833,-176.517,7.963,148.530
C06005=1182.830,321.578,-72.801,-176.519,7.960,148.530
C06006=1182.834,321.330,-72.770,-176.522,7.958,148.530
C06007=1182.839,321.082,-72.739,-176.524,7.955,148.530
C06008=1182.843,320.833,-72.706,-176.526,7.952,148.530
C06009=1182.848,320.585,-72.676,-176.529,7.948,148.530
C06010=1182.851,320.337,-72.644,-176.531,7.945,148.530
C06011=1182.856,320.089,-72.613,-176.534,7.942,148.530
C06012=1182.860,319.841,-72.581,-176.536,7.939,148.530
C06013=1182.864,319.594,-72.550,-176.539,7.936,148.530
C06014=1182.868,319.345,-72.519,-176.541,7.933,148.529
C06015=1182.872,319.098,-72.487,-176.544,7.930,148.529
C06016=1182.876,318.849,-72.456,-176.546,7.926,148.529
C06017=1182.881,318.601,-72.425,-176.549,7.923,148.529
C06018=1182.885,318.353,-72.393,-176.551,7.921,148.529
C06019=1182.889,318.105,-72.363,-176.554,7.918,148.529
C06020=1182.893,317.857,-72.331,-176.556,7.915,148.529
C06021=1182.898,317.609,-72.300,-176.558,7.912,148.529
C06022=1182.902,317.362,-72.268,-176.561,7.909,148.529
C06023=1182.906,317.113,-72.237,-176.564,7.906,148.529
C06024=1182.910,316.865,-72.207,-176.566,7.902,148.529
C06025=1182.914,316.617,-72.175,-176.569,7.899,148.529
C06026=1182.919,316.369,-72.144,-176.571,7.896,148.528
C06027=1182.922,316.121,-72.113,-176.574,7.893,148.528
C06028=1182.926,315.874,-72.082,-176.577,7.890,148.528
C06029=1182.931,315.626,-72.051,-176.578,7.887,148.528
C06030=1182.935,315.377,-72.020,-176.581,7.884,148.528
C06031=1182.939,315.130,-71.989,-176.584,7.881,148.528
C06032=1182.943,314.881,-71.957,-176.586,7.878,148.528
C06033=1182.948,314.605,-71.923,-176.589,7.875,148.528
C06034=1182.953,314.328,-71.889,-176.592,7.871,148.528
C06035=1182.958,314.051,-71.854,-176.594,7.868,148.528
C06036=1182.962,313.775,-71.819,-176.597,7.864,148.528
C06037=1182.966,313.527,-71.789,-176.600,7.862,148.528
C06038=1182.971,313.279,-71.758,-176.602,7.859,148.528
C06039=1182.975,313.030,-71.727,-176.605,7.856,148.528
C06040=1182.980,312.782,-71.696,-176.607,7.853,148.528
C06041=1182.984,312.534,-71.665,-176.610,7.850,148.528
C06042=1182.987,312.287,-71.634,-176.612,7.846,148.528
C06043=1182.992,312.039,-71.603,-176.615,7.843,148.528
C06044=1182.996,311.791,-71.572,-176.618,7.840,148.528
C06045=1183.000,311.542,-71.541,-176.620,7.837,148.527
C06046=1183.004,311.294,-71.511,-176.622,7.835,148.527
C06047=1183.009,311.046,-71.480,-176.625,7.832,148.527
C06048=1183.013,310.798,-71.449,-176.627,7.829,148.527
C06049=1183.017,310.550,-71.418,-176.630,7.826,148.527
C06050=1183.021,310.302,-71.388,-176.633,7.823,148.527
C06051=1183.025,310.053,-71.357,-176.635,7.819,148.527
C06052=1183.030,309.806,-71.326,-176.638,7.816,148.527
C06053=1183.035,309.558,-71.296,-176.640,7.813,148.527
C06054=1183.038,309.310,-71.265,-176.642,7.811,148.527
C06055=1183.042,309.061,-71.234,-176.645,7.808,148.527
C06056=1183.047,308.813,-71.204,-176.647,7.805,148.527
C06057=1183.051,308.566,-71.173,-176.650,7.802,148.527
C06058=1183.055,308.317,-71.142,-176.653,7.799,148.527
C06059=1183.060,308.069,-71.111,-176.655,7.795,148.527
C06060=1183.063,307.821,-71.081,-176.658,7.792,148.527
C06061=1183.068,307.573,-71.051,-176.661,7.789,148.527
C06062=1183.073,307.325,-71.020,-176.662,7.787,148.527
C06063=1183.076,307.077,-70.990,-176.665,7.784,148.527
C06064=1183.081,306.829,-70.959,-176.668,7.781,148.527
C06065=1183.085,306.581,-70.929,-176.670,7.778,148.527
C06066=1183.089,306.333,-70.898,-176.673,7.775,148.527
C06067=1183.093,306.084,-70.867,-176.675,7.772,148.527
C06068=1183.098,305.836,-70.838,-176.678,7.769,148.527
C06069=1183.102,305.588,-70.807,-176.680,7.767,148.527
C06070=1183.106,305.340,-70.777,-176.683,7.764,148.527
C06071=1183.111,305.092,-70.746,-176.685,7.760,148.527
C06072=1183.115,304.843,-70.716,-176.688,7.757,148.527
C06073=1183.119,304.596,-70.685,-176.691,7.754,148.527
C06074=1183.123,304.348,-70.655,-176.693,7.751,148.527
C06075=1183.127,304.100,-70.624,-176.696,7.748,148.526
C06076=1183.132,303.851,-70.594,-176.698,7.746,148.526
C06077=1183.136,303.604,-70.564,-176.700,7.743,148.526
C06078=1183.140,303.355,-70.533,-176.703,7.740,148.527
C06079=1183.144,303.107,-70.504,-176.706,7.737,148.527
C06080=1183.149,302.859,-70.473,-176.708,7.733,148.526
C06081=1183.153,302.611,-70.443,-176.711,7.730,148.526
C06082=1183.158,302.363,-70.413,-176.713,7.728,148.526
C06083=1183.162,302.115,-70.383,-176.716,7.725,148.526
C06084=1183.167,301.866,-70.352,-176.718,7.722,148.526
C06085=1183.170,301.618,-70.322,-176.721,7.719,148.526
C06086=1183.174,301.370,-70.292,-176.723,7.716,148.526
C06087=1183.179,301.122,-70.262,-176.726,7.713,148.526
C06088=1183.183,300.874,-70.232,-176.729,7.710,148.526
C06089=1183.187,300.626,-70.201,-176.731,7.708,148.526
C06090=1183.192,300.377,-70.172,-176.733,7.705,148.526
C06091=1183.195,300.130,-70.142,-176.736,7.702,148.526
C06092=1183.200,299.881,-70.112,-176.739,7.699,148.526
C06093=1183.204,299.633,-70.082,-176.741,7.696,148.526
C06094=1183.209,299.385,-70.052,-176.744,7.693,148.526
C06095=1183.213,299.137,-70.021,-176.746,7.690,148.526
C06096=1183.217,298.888,-69.992,-176.749,7.687,148.526
C06097=1183.221,298.640,-69.961,-176.751,7.684,148.526
C06098=1183.225,298.392,-69.931,-176.754,7.681,148.526
C06099=1183.230,298.144,-69.902,-176.757,7.678,148.526
C06100=1183.234,297.896,-69.871,-176.759,7.676,148.526
C06101=1183.238,297.648,-69.842,-176.762,7.673,148.526
C06102=1183.243,297.399,-69.812,-176.764,7.670,148.526
C06103=1183.246,297.152,-69.782,-176.767,7.667,148.526
C06104=1183.251,296.903,-69.752,-176.769,7.664,148.526
C06105=1183.256,296.655,-69.723,-176.772,7.661,148.526
C06106=1183.259,296.407,-69.692,-176.774,7.658,148.526
C06107=1183.264,296.159,-69.663,-176.777,7.655,148.526
C06108=1183.269,295.910,-69.633,-176.780,7.652,148.526
C06109=1183.272,295.663,-69.603,-176.782,7.649,148.526
C06110=1183.277,295.414,-69.573,-176.785,7.646,148.526
C06111=1183.281,295.166,-69.544,-176.787,7.644,148.526
C06112=1183.286,294.918,-69.514,-176.790,7.641,148.526
C06113=1183.290,294.670,-69.484,-176.792,7.638,148.526
C06114=1183.294,294.422,-69.454,-176.795,7.635,148.526
C06115=1183.298,294.173,-69.425,-176.798,7.632,148.526
C06116=1183.302,293.925,-69.395,-176.800,7.630,148.526
C06117=1183.307,293.676,-69.365,-176.803,7.627,148.526
C06118=1183.311,293.428,-69.336,-176.805,7.624,148.526
C06119=1183.315,293.180,-69.306,-176.808,7.621,148.526
C06120=1183.319,292.932,-69.276,-176.810,7.618,148.526
C06121=1183.323,292.684,-69.247,-176.812,7.615,148.526
C06122=1183.328,292.436,-69.217,-176.815,7.612,148.526
C06123=1183.332,292.188,-69.188,-176.818,7.609,148.526
C06124=1183.336,291.939,-69.158,-176.821,7.606,148.526
C06125=1183.341,291.691,-69.128,-176.823,7.603,148.527
C06126=1183.346,291.443,-69.099,-176.825,7.601,148.527
C06127=1183.350,291.195,-69.070,-176.828,7.598,148.527
C06128=1183.354,290.947,-69.040,-176.831,7.595,148.527
C06129=1183.358,290.698,-69.011,-176.834,7.592,148.527
C06130=1183.362,290.450,-68.981,-176.836,7.590,148.527
C06131=1183.367,290.202,-68.952,-176.838,7.587,148.527
C06132=1183.371,289.953,-68.922,-176.841,7.584,148.527
C06133=1183.375,289.705,-68.893,-176.844,7.581,148.527
C06134=1183.379,289.457,-68.864,-176.846,7.578,148.527
C06135=1183.383,289.209,-68.834,-176.848,7.576,148.527
C06136=1183.388,288.961,-68.805,-176.851,7.573,148.527
C06137=1183.393,288.686,-68.772,-176.854,7.570,148.527
C06138=1183.398,288.412,-68.740,-176.857,7.566,148.527
C06139=1183.403,288.137,-68.707,-176.860,7.563,148.527
C06140=1183.407,287.862,-68.676,-176.863,7.560,148.527
C06141=1183.412,287.614,-68.646,-176.865,7.557,148.527
C06142=1183.416,287.366,-68.617,-176.867,7.555,148.527
C06143=1183.420,287.117,-68.587,-176.870,7.552,148.527
C06144=1183.424,286.869,-68.558,-176.873,7.549,148.527
C06145=1183.429,286.620,-68.529,-176.876,7.546,148.527
C06146=1183.433,286.373,-68.500,-176.878,7.544,148.527
C06147=1183.438,286.124,-68.471,-176.880,7.541,148.527
C06148=1183.442,285.876,-68.441,-176.883,7.538,148.527
C06149=1183.446,285.627,-68.413,-176.886,7.535,148.527
C06150=1183.450,285.379,-68.383,-176.888,7.532,148.527
C06151=1183.454,285.132,-68.355,-176.891,7.529,148.527
C06152=1183.459,284.884,-68.325,-176.894,7.526,148.527
C06153=1183.463,284.635,-68.296,-176.896,7.523,148.527
C06154=1183.467,284.386,-68.267,-176.898,7.521,148.527
C06155=1183.472,284.139,-68.238,-176.901,7.518,148.527
C06156=1183.477,283.890,-68.209,-176.904,7.515,148.528
C06157=1183.481,283.642,-68.180,-176.907,7.512,148.528
C06158=1183.484,283.394,-68.151,-176.909,7.510,148.528
C06159=1183.489,283.145,-68.122,-176.911,7.507,148.528
C06160=1183.493,282.897,-68.093,-176.914,7.504,148.528
C06161=1183.498,282.648,-68.064,-176.917,7.501,148.528
C06162=1183.502,282.400,-68.035,-176.919,7.499,148.528
C06163=1183.506,282.152,-68.007,-176.922,7.496,148.528
C06164=1183.511,281.904,-67.978,-176.925,7.493,148.528
C06165=1183.515,281.655,-67.949,-176.927,7.490,148.528
C06166=1183.519,281.407,-67.919,-176.929,7.488,148.528
C06167=1183.524,281.159,-67.890,-176.932,7.485,148.528
C06168=1183.528,280.911,-67.862,-176.935,7.482,148.528
C06169=1183.532,280.662,-67.833,-176.937,7.480,148.528
C06170=1183.537,280.414,-67.804,-176.940,7.477,148.528
C06171=1183.541,280.166,-67.776,-176.942,7.474,148.528
C06172=1183.545,279.917,-67.747,-176.945,7.471,148.528
C06173=1183.550,279.669,-67.718,-176.947,7.469,148.528
C06174=1183.554,279.421,-67.689,-176.950,7.466,148.528
C06175=1183.558,279.172,-67.661,-176.953,7.463,148.528
C06176=1183.562,278.924,-67.631,-176.956,7.460,148.528
C06177=1183.567,278.676,-67.603,-176.958,7.458,148.529
C06178=1183.571,278.427,-67.575,-176.960,7.455,148.529
C06179=1183.575,278.179,-67.545,-176.963,7.452,148.529
C06180=1183.580,277.931,-67.517,-176.966,7.450,148.529
C06181=1183.584,277.682,-67.489,-176.969,7.447,148.529
C06182=1183.589,277.435,-67.460,-176.971,7.444,148.529
C06183=1183.593,277.186,-67.432,-176.973,7.442,148.529
C06184=1183.597,276.937,-67.403,-176.976,7.439,148.529
C06185=1183.602,276.690,-67.374,-176.979,7.436,148.529
C06186=1183.606,276.441,-67.346,-176.982,7.433,148.529
C06187=1183.610,276.192,-67.317,-176.984,7.430,148.529
C06188=1183.614,275.944,-67.289,-176.986,7.427,148.529
C06189=1183.619,275.696,-67.260,-176.989,7.424,148.529
C06190=1183.623,275.448,-67.232,-176.991,7.422,148.529
C06191=1183.627,275.199,-67.203,-176.994,7.419,148.529
C06192=1183.632,274.950,-67.174,-176.997,7.416,148.530
C06193=1183.636,274.703,-67.147,-176.999,7.414,148.530
C06194=1183.641,274.454,-67.118,-177.002,7.411,148.530
C06195=1183.645,274.206,-67.089,-177.005,7.409,148.530
C06196=1183.649,273.957,-67.061,-177.008,7.406,148.530
C06197=1183.654,273.710,-67.033,-177.010,7.403,148.530
C06198=1183.658,273.461,-67.004,-177.013,7.400,148.530
C06199=1183.662,273.212,-66.976,-177.015,7.397,148.530
C06200=1183.667,272.964,-66.948,-177.017,7.395,148.530
C06201=1183.671,272.715,-66.919,-177.020,7.392,148.530
C06202=1183.676,272.467,-66.891,-177.023,7.389,148.530
C06203=1183.680,272.219,-66.863,-177.025,7.387,148.530
C06204=1183.684,271.971,-66.835,-177.028,7.384,148.530
C06205=1183.688,271.722,-66.806,-177.031,7.381,148.531
C06206=1183.693,271.474,-66.779,-177.033,7.379,148.531
C06207=1183.697,271.225,-66.750,-177.036,7.376,148.531
C06208=1183.702,270.977,-66.722,-177.039,7.373,148.531
C06209=1183.706,270.728,-66.693,-177.041,7.371,148.531
C06210=1183.710,270.480,-66.666,-177.043,7.368,148.531
C06211=1183.714,270.232,-66.638,-177.046,7.365,148.531
C06212=1183.719,269.984,-66.609,-177.048,7.363,148.531
C06213=1183.723,269.735,-66.581,-177.052,7.360,148.531
C06214=1183.728,269.487,-66.553,-177.054,7.357,148.531
C06215=1183.732,269.238,-66.524,-177.056,7.355,148.531
C06216=1183.736,268.990,-66.497,-177.059,7.352,148.532
C06217=1183.741,268.742,-66.468,-177.062,7.349,148.532
C06218=1183.745,268.494,-66.440,-177.064,7.347,148.532
C06219=1183.749,268.245,-66.413,-177.067,7.344,148.532
C06220=1183.754,267.996,-66.384,-177.069,7.342,148.532
C06221=1183.759,267.748,-66.357,-177.072,7.339,148.532
C06222=1183.762,267.500,-66.328,-177.075,7.336,148.532
C06223=1183.767,267.252,-66.300,-177.077,7.334,148.532
C06224=1183.771,267.003,-66.272,-177.080,7.331,148.532
C06225=1183.776,266.755,-66.245,-177.082,7.328,148.532
C06226=1183.780,266.507,-66.217,-177.085,7.326,148.532
C06227=1183.785,266.258,-66.188,-177.088,7.323,148.533
C06228=1183.789,266.010,-66.161,-177.091,7.320,148.533
C06229=1183.793,265.761,-66.133,-177.093,7.318,148.533
C06230=1183.797,265.513,-66.105,-177.095,7.315,148.533
C06231=1183.803,265.265,-66.077,-177.098,7.313,148.533
C06232=1183.807,265.016,-66.050,-177.100,7.310,148.533
C06233=1183.811,264.768,-66.022,-177.104,7.307,148.533
C06234=1183.815,264.519,-65.994,-177.106,7.305,148.533
C06235=1183.819,264.271,-65.967,-177.108,7.302,148.533
C06236=1183.824,264.022,-65.938,-177.111,7.299,148.533
C06237=1183.828,263.774,-65.910,-177.113,7.297,148.533
C06238=1183.833,263.525,-65.883,-177.117,7.294,148.534
C06239=1183.837,263.277,-65.855,-177.119,7.292,148.534
C06240=1183.841,263.028,-65.828,-177.121,7.289,148.534
C06241=1183.846,262.756,-65.798,-177.124,7.286,148.534
C06242=1183.851,262.482,-65.767,-177.127,7.284,148.534
C06243=1183.856,262.210,-65.737,-177.130,7.281,148.534
C06244=1183.861,261.936,-65.706,-177.133,7.278,148.534
C06245=1183.865,261.688,-65.678,-177.135,7.276,148.534
C06246=1183.870,261.440,-65.651,-177.138,7.273,148.535
C06247=1183.874,261.191,-65.623,-177.141,7.270,148.535
C06248=1183.879,260.943,-65.596,-177.143,7.268,148.535
C06249=1183.883,260.695,-65.568,-177.146,7.265,148.535
C06250=1183.887,260.446,-65.541,-177.148,7.263,148.535
C06251=1183.891,260.198,-65.513,-177.151,7.260,148.535
C06252=1183.896,259.949,-65.486,-177.154,7.257,148.535
C06253=1183.900,259.701,-65.458,-177.156,7.255,148.535
C06254=1183.904,259.452,-65.431,-177.159,7.252,148.536
C06255=1183.909,259.204,-65.404,-177.161,7.250,148.536
C06256=1183.913,258.956,-65.376,-177.164,7.247,148.536
C06257=1183.917,258.707,-65.348,-177.167,7.244,148.536
C06258=1183.922,258.458,-65.321,-177.169,7.242,148.536
C06259=1183.926,258.210,-65.293,-177.172,7.239,148.536
C06260=1183.931,257.962,-65.266,-177.174,7.237,148.536
C06261=1183.935,257.713,-65.239,-177.177,7.234,148.536
C06262=1183.939,257.465,-65.211,-177.179,7.232,148.536
C06263=1183.944,257.216,-65.184,-177.183,7.229,148.537
C06264=1183.949,256.968,-65.157,-177.185,7.226,148.537
C06265=1183.953,256.719,-65.129,-177.187,7.224,148.537
C06266=1183.957,256.471,-65.102,-177.190,7.221,148.537
C06267=1183.962,256.222,-65.075,-177.193,7.219,148.537
C06268=1183.966,255.974,-65.048,-177.196,7.216,148.537
C06269=1183.971,255.726,-65.020,-177.198,7.214,148.537
C06270=1183.975,255.477,-64.993,-177.201,7.212,148.538
C06271=1183.980,255.228,-64.965,-177.204,7.209,148.538
C06272=1183.984,254.980,-64.938,-177.206,7.206,148.538
C06273=1183.988,254.732,-64.912,-177.209,7.203,148.538
C06274=1183.993,254.483,-64.885,-177.211,7.202,148.538
C06275=1183.997,254.235,-64.857,-177.214,7.199,148.538
C06276=1184.001,253.986,-64.830,-177.216,7.196,148.538
C06277=1184.006,253.738,-64.803,-177.219,7.194,148.539
C06278=1184.011,253.489,-64.776,-177.221,7.192,148.539
C06279=1184.015,253.241,-64.749,-177.224,7.189,148.539
C06280=1184.019,252.992,-64.722,-177.226,7.187,148.539
C06281=1184.024,252.744,-64.695,-177.230,7.184,148.539
C06282=1184.028,252.495,-64.668,-177.232,7.181,148.539
C06283=1184.032,252.246,-64.640,-177.234,7.179,148.539
C06284=1184.037,251.998,-64.613,-177.238,7.176,148.539
C06285=1184.041,251.749,-64.587,-177.240,7.174,148.540
C06286=1184.046,251.501,-64.560,-177.243,7.171,148.540
C06287=1184.050,251.252,-64.533,-177.245,7.169,148.540
C06288=1184.055,251.004,-64.506,-177.248,7.166,148.540
C06289=1184.059,250.756,-64.479,-177.250,7.164,148.540
C06290=1184.064,250.507,-64.452,-177.253,7.161,148.540
C06291=1184.068,250.258,-64.425,-177.255,7.159,148.540
C06292=1184.072,250.010,-64.398,-177.258,7.156,148.541
C06293=1184.076,249.761,-64.371,-177.261,7.154,148.541
C06294=1184.081,249.513,-64.344,-177.264,7.151,148.541
C06295=1184.086,249.264,-64.317,-177.266,7.149,148.541
C06296=1184.089,249.016,-64.291,-177.269,7.147,148.541
C06297=1184.094,248.768,-64.264,-177.271,7.144,148.541
C06298=1184.099,248.519,-64.237,-177.274,7.141,148.541
C06299=1184.104,248.270,-64.210,-177.277,7.140,148.542
C06300=1184.108,248.022,-64.184,-177.279,7.137,148.542
C06301=1184.112,247.773,-64.157,-177.281,7.135,148.542
C06302=1184.117,247.525,-64.130,-177.285,7.132,148.542
C06303=1184.121,247.277,-64.103,-177.287,7.130,148.542
C06304=1184.126,247.028,-64.077,-177.290,7.127,148.542
C06305=1184.130,246.779,-64.050,-177.292,7.125,148.543
C06306=1184.134,246.531,-64.023,-177.295,7.122,148.543
C06307=1184.139,246.282,-63.996,-177.297,7.120,148.543
C06308=1184.143,246.034,-63.971,-177.300,7.117,148.543
C06309=1184.148,245.785,-63.943,-177.302,7.115,148.543
C06310=1184.152,245.537,-63.917,-177.306,7.112,148.543
C06311=1184.157,245.289,-63.890,-177.308,7.110,148.544
C06312=1184.161,245.039,-63.864,-177.311,7.107,148.544
C06313=1184.165,244.791,-63.837,-177.313,7.105,148.544
C06314=1184.170,244.543,-63.810,-177.316,7.102,148.544
C06315=1184.174,244.294,-63.784,-177.319,7.101,148.544
C06316=1184.179,244.045,-63.757,-177.321,7.098,148.544
C06317=1184.183,243.797,-63.731,-177.324,7.095,148.544
C06318=1184.188,243.548,-63.704,-177.327,7.093,148.545
C06319=1184.192,243.300,-63.678,-177.329,7.091,148.545
C06320=1184.197,243.051,-63.652,-177.332,7.088,148.545
C06321=1184.201,242.803,-63.625,-177.334,7.086,148.545
C06322=1184.205,242.554,-63.598,-177.337,7.083,148.545
C06323=1184.209,242.305,-63.572,-177.340,7.081,148.546
C06324=1184.214,242.057,-63.545,-177.342,7.078,148.546
C06325=1184.218,241.808,-63.520,-177.345,7.076,148.546
C06326=1184.223,241.560,-63.492,-177.347,7.074,148.546
C06327=1184.227,241.311,-63.467,-177.350,7.071,148.546
C06328=1184.233,241.063,-63.440,-177.353,7.069,148.547
C06329=1184.237,240.814,-63.414,-177.355,7.066,148.547
C06330=1184.241,240.566,-63.388,-177.358,7.065,148.547
C06331=1184.246,240.317,-63.361,-177.361,7.062,148.547
C06332=1184.250,240.069,-63.335,-177.363,7.060,148.547
C06333=1184.255,239.820,-63.309,-177.366,7.057,148.547
C06334=1184.259,239.571,-63.283,-177.368,7.055,148.547
C06335=1184.263,239.323,-63.256,-177.371,7.052,148.548
C06336=1184.268,239.073,-63.230,-177.374,7.050,148.548
C06337=1184.272,238.826,-63.204,-177.376,7.048,148.548
C06338=1184.277,238.577,-63.178,-177.379,7.045,148.548
C06339=1184.281,238.328,-63.152,-177.382,7.043,148.549
C06340=1184.285,238.080,-63.125,-177.384,7.040,148.549
C06341=1184.290,237.831,-63.099,-177.387,7.038,148.549
C06342=1184.294,237.582,-63.073,-177.390,7.035,148.549
C06343=1184.299,237.334,-63.047,-177.392,7.033,148.549
C06344=1184.304,237.085,-63.021,-177.395,7.031,148.549
C06345=1184.309,236.813,-62.993,-177.398,7.029,148.550
C06346=1184.313,236.542,-62.964,-177.401,7.026,148.550
C06347=1184.318,236.270,-62.936,-177.404,7.023,148.550
C06348=1184.323,235.999,-62.907,-177.406,7.021,148.550
C06349=1184.328,235.751,-62.881,-177.409,7.018,148.550
C06350=1184.332,235.502,-62.856,-177.411,7.016,148.551
C06351=1184.336,235.254,-62.829,-177.415,7.014,148.551
C06352=1184.341,235.004,-62.803,-177.417,7.011,148.551
C06353=1184.346,234.756,-62.777,-177.419,7.010,148.551
C06354=1184.350,234.508,-62.752,-177.422,7.007,148.551
C06355=1184.354,234.259,-62.726,-177.425,7.005,148.552
C06356=1184.359,234.010,-62.699,-177.427,7.002,148.552
C06357=1184.363,233.761,-62.673,-177.430,7.000,148.552
C06358=1184.368,233.513,-62.648,-177.432,6.998,148.552
C06359=1184.372,233.265,-62.622,-177.436,6.995,148.552
C06360=1184.376,233.016,-62.596,-177.438,6.993,148.553
C06361=1184.380,232.767,-62.570,-177.441,6.991,148.553
C06362=1184.386,232.518,-62.544,-177.443,6.988,148.553
C06363=1184.390,232.270,-62.519,-177.446,6.987,148.553
C06364=1184.394,232.021,-62.493,-177.448,6.984,148.553
C06365=1184.399,231.773,-62.468,-177.451,6.982,148.554
C06366=1184.403,231.524,-62.442,-177.454,6.979,148.554
C06367=1184.408,231.275,-62.416,-177.456,6.977,148.554
C06368=1184.412,231.026,-62.390,-177.459,6.975,148.554
C06369=1184.417,230.778,-62.364,-177.462,6.972,148.554
C06370=1184.422,230.529,-62.339,-177.464,6.970,148.555
C06371=1184.426,230.280,-62.313,-177.467,6.967,148.555
C06372=1184.431,230.032,-62.287,-177.470,6.966,148.555
C06373=1184.435,229.783,-62.262,-177.472,6.963,148.555
C06374=1184.439,229.535,-62.236,-177.475,6.961,148.556
C06375=1184.444,229.287,-62.211,-177.477,6.959,148.556
C06376=1184.448,229.038,-62.185,-177.480,6.957,148.556
C06377=1184.452,228.789,-62.159,-177.483,6.954,148.556
C06378=1184.457,228.541,-62.134,-177.486,6.952,148.556
C06379=1184.462,228.292,-62.108,-177.488,6.949,148.557
C06380=1184.466,228.043,-62.083,-177.491,6.947,148.557
C06381=1184.471,227.794,-62.057,-177.494,6.945,148.557
C06382=1184.475,227.546,-62.032,-177.496,6.942,148.557
C06383=1184.479,227.297,-62.006,-177.499,6.941,148.558
C06384=1184.484,227.049,-61.981,-177.501,6.939,148.558
C06385=1184.488,226.800,-61.955,-177.504,6.936,148.558
C06386=1184.493,226.551,-61.930,-177.507,6.934,148.558
C06387=1184.498,226.302,-61.904,-177.509,6.932,148.558
C06388=1184.502,226.054,-61.879,-177.512,6.929,148.559
C06389=1184.507,225.806,-61.853,-177.515,6.927,148.559
C06390=1184.511,225.556,-61.828,-177.517,6.925,148.559
C06391=1184.516,225.307,-61.802,-177.520,6.922,148.559
C06392=1184.520,225.059,-61.777,-177.523,6.921,148.560
C06393=1184.525,224.810,-61.751,-177.525,6.918,148.560
C06394=1184.530,224.562,-61.727,-177.528,6.916,148.560
C06395=1184.534,224.313,-61.701,-177.531,6.914,148.560
C06396=1184.538,224.064,-61.675,-177.533,6.911,148.560
C06397=1184.543,223.816,-61.651,-177.536,6.909,148.561
C06398=1184.547,223.567,-61.625,-177.538,6.907,148.561
C06399=1184.552,223.319,-61.600,-177.541,6.904,148.561
C06400=1184.556,223.069,-61.575,-177.544,6.903,148.561
C06401=1184.561,222.821,-61.550,-177.546,6.900,148.562
C06402=1184.565,222.572,-61.524,-177.550,6.898,148.562
C06403=1184.570,222.324,-61.499,-177.552,6.896,148.562
C06404=1184.574,222.075,-61.474,-177.554,6.894,148.562
C06405=1184.578,221.826,-61.449,-177.558,6.891,148.563
C06406=1184.583,221.578,-61.424,-177.560,6.889,148.563
C06407=1184.588,221.328,-61.399,-177.562,6.887,148.563
C06408=1184.593,221.080,-61.373,-177.566,6.885,148.563
C06409=1184.597,220.831,-61.348,-177.568,6.882,148.563
C06410=1184.601,220.583,-61.323,-177.570,6.881,148.564
C06411=1184.606,220.333,-61.298,-177.573,6.879,148.564
C06412=1184.611,220.085,-61.273,-177.576,6.876,148.564
C06413=1184.615,219.836,-61.248,-177.578,6.874,148.565
C06414=1184.619,219.588,-61.223,-177.581,6.872,148.565
C06415=1184.624,219.339,-61.198,-177.584,6.869,148.565
C06416=1184.628,219.091,-61.173,-177.587,6.868,148.565
C06417=1184.633,218.841,-61.148,-177.589,6.865,148.565
C06418=1184.637,218.593,-61.123,-177.592,6.863,148.566
C06419=1184.642,218.344,-61.098,-177.595,6.861,148.566
C06420=1184.647,218.095,-61.073,-177.597,6.859,148.566
C06421=1184.651,217.847,-61.048,-177.600,6.856,148.566
C06422=1184.655,217.598,-61.023,-177.602,6.854,148.567
C06423=1184.661,217.349,-60.999,-177.605,6.852,148.567
C06424=1184.664,217.101,-60.973,-177.607,6.850,148.567
C06425=1184.669,216.852,-60.949,-177.610,6.847,148.567
C06426=1184.674,216.603,-60.924,-177.613,6.846,148.568
C06427=1184.678,216.355,-60.899,-177.616,6.844,148.568
C06428=1184.683,216.106,-60.874,-177.618,6.841,148.568
C06429=1184.687,215.857,-60.849,-177.621,6.839,148.568
C06430=1184.692,215.609,-60.824,-177.624,6.837,148.569
C06431=1184.696,215.360,-60.799,-177.626,6.835,148.569
C06432=1184.701,215.111,-60.775,-177.629,6.832,148.569
C06433=1184.705,214.862,-60.750,-177.632,6.831,148.570
C06434=1184.710,214.614,-60.725,-177.634,6.829,148.570
C06435=1184.714,214.365,-60.701,-177.637,6.826,148.570
C06436=1184.719,214.116,-60.676,-177.640,6.824,148.570
C06437=1184.723,213.867,-60.652,-177.642,6.822,148.571
C06438=1184.728,213.619,-60.627,-177.645,6.820,148.571
C06439=1184.732,213.370,-60.601,-177.648,6.817,148.571
C06440=1184.737,213.121,-60.577,-177.650,6.816,148.571
C06441=1184.741,212.872,-60.552,-177.653,6.814,148.572
C06442=1184.746,212.624,-60.528,-177.655,6.812,148.572
C06443=1184.751,212.375,-60.503,-177.658,6.809,148.572
C06444=1184.755,212.126,-60.479,-177.661,6.807,148.572
C06445=1184.760,211.877,-60.454,-177.663,6.805,148.573
C06446=1184.764,211.629,-60.430,-177.667,6.803,148.573
C06447=1184.769,211.379,-60.405,-177.669,6.801,148.573
C06448=1184.773,211.131,-60.380,-177.671,6.799,148.573
C06449=1184.778,210.861,-60.354,-177.675,6.796,148.574
C06450=1184.783,210.590,-60.328,-177.677,6.794,148.574
C06451=1184.788,210.320,-60.301,-177.680,6.792,148.574
C06452=1184.793,210.049,-60.274,-177.683,6.790,148.575
C06453=1184.798,209.801,-60.250,-177.685,6.788,148.575
C06454=1184.802,209.552,-60.225,-177.689,6.785,148.575
C06455=1184.806,209.303,-60.201,-177.691,6.783,148.575
C06456=1184.812,209.054,-60.176,-177.694,6.781,148.576
C06457=1184.816,208.806,-60.152,-177.696,6.779,148.576
C06458=1184.820,208.557,-60.128,-177.699,6.777,148.576
C06459=1184.825,208.308,-60.103,-177.702,6.775,148.577
C06460=1184.830,208.059,-60.080,-177.704,6.773,148.577
C06461=1184.835,207.810,-60.055,-177.707,6.771,148.577
C06462=1184.839,207.561,-60.030,-177.710,6.768,148.577
C06463=1184.843,207.313,-60.006,-177.713,6.766,148.578
C06464=1184.848,207.064,-59.982,-177.715,6.764,148.578
C06465=1184.852,206.816,-59.958,-177.718,6.762,148.578
C06466=1184.856,206.567,-59.933,-177.721,6.760,148.578
C06467=1184.861,206.318,-59.909,-177.723,6.758,148.579
C06468=1184.866,206.069,-59.885,-177.726,6.756,148.579
C06469=1184.871,205.820,-59.861,-177.728,6.754,148.579
C06470=1184.875,205.571,-59.836,-177.731,6.752,148.580
C06471=1184.879,205.323,-59.812,-177.734,6.750,148.580
C06472=1184.884,205.074,-59.788,-177.736,6.748,148.580
C06473=1184.889,204.825,-59.764,-177.739,6.746,148.580
C06474=1184.894,204.576,-59.740,-177.742,6.744,148.581
C06475=1184.897,204.327,-59.715,-177.744,6.742,148.581
C06476=1184.903,204.079,-59.691,-177.747,6.739,148.581
C06477=1184.907,203.830,-59.667,-177.750,6.737,148.581
C06478=1184.912,203.581,-59.643,-177.752,6.736,148.582
C06479=1184.916,203.333,-59.619,-177.755,6.734,148.582
C06480=1184.921,203.083,-59.595,-177.757,6.732,148.582
C06481=1184.925,202.834,-59.571,-177.760,6.729,148.583
C06482=1184.930,202.586,-59.547,-177.763,6.727,148.583
C06483=1184.934,202.337,-59.523,-177.766,6.725,148.583
C06484=1184.939,202.088,-59.499,-177.768,6.724,148.584
C06485=1184.944,201.840,-59.475,-177.771,6.722,148.584
C06486=1184.949,201.591,-59.451,-177.774,6.719,148.584
C06487=1184.953,201.342,-59.427,-177.777,6.717,148.584
C06488=1184.957,201.093,-59.404,-177.779,6.715,148.585
C06489=1184.961,200.844,-59.379,-177.781,6.713,148.585
C06490=1184.966,200.596,-59.355,-177.784,6.711,148.585
C06491=1184.971,200.346,-59.331,-177.787,6.709,148.586
C06492=1184.976,200.098,-59.307,-177.790,6.707,148.586
C06493=1184.980,199.849,-59.284,-177.793,6.705,148.586
C06494=1184.985,199.601,-59.260,-177.795,6.703,148.586
C06495=1184.990,199.351,-59.237,-177.797,6.701,148.587
C06496=1184.994,199.103,-59.212,-177.800,6.699,148.587
C06497=1184.998,198.853,-59.189,-177.803,6.697,148.587
C06498=1185.002,198.605,-59.165,-177.806,6.695,148.588
C06499=1185.008,198.356,-59.141,-177.808,6.693,148.588
C06500=1185.012,198.107,-59.117,-177.811,6.691,148.588
C06501=1185.017,197.858,-59.093,-177.813,6.689,148.589
C06502=1185.021,197.610,-59.069,-177.816,6.687,148.589
C06503=1185.026,197.361,-59.046,-177.819,6.685,148.589
C06504=1185.031,197.112,-59.023,-177.822,6.683,148.589
C06505=1185.035,196.863,-58.998,-177.824,6.681,148.590
C06506=1185.040,196.614,-58.975,-177.827,6.679,148.590
C06507=1185.044,196.366,-58.951,-177.830,6.677,148.590
C06508=1185.049,196.117,-58.928,-177.832,6.676,148.591
C06509=1185.054,195.868,-58.904,-177.835,6.673,148.591
C06510=1185.058,195.619,-58.880,-177.838,6.671,148.591
C06511=1185.063,195.370,-58.857,-177.840,6.669,148.592
C06512=1185.067,195.121,-58.834,-177.843,6.667,148.592
C06513=1185.072,194.873,-58.809,-177.846,6.665,148.592
C06514=1185.076,194.624,-58.786,-177.848,6.664,148.593
C06515=1185.081,194.375,-58.763,-177.850,6.661,148.593
C06516=1185.086,194.126,-58.739,-177.854,6.659,148.593
C06517=1185.090,193.877,-58.715,-177.856,6.657,148.593
C06518=1185.095,193.628,-58.692,-177.859,6.655,148.594
C06519=1185.100,193.379,-58.669,-177.862,6.653,148.594
C06520=1185.104,193.130,-58.645,-177.864,6.652,148.594
C06521=1185.109,192.882,-58.621,-177.867,6.650,148.595
C06522=1185.113,192.633,-58.598,-177.869,6.648,148.595
C06523=1185.118,192.384,-58.574,-177.872,6.646,148.595
C06524=1185.122,192.135,-58.552,-177.875,6.643,148.596
C06525=1185.127,191.886,-58.528,-177.878,6.642,148.596
C06526=1185.132,191.637,-58.505,-177.880,6.640,148.596
C06527=1185.136,191.389,-58.481,-177.883,6.638,148.597
C06528=1185.141,191.140,-58.457,-177.885,6.636,148.597
C06529=1185.145,190.890,-58.434,-177.888,6.634,148.597
C06530=1185.150,190.641,-58.411,-177.891,6.632,148.598
C06531=1185.155,190.392,-58.387,-177.893,6.630,148.598
C06532=1185.159,190.144,-58.365,-177.897,6.628,148.598
C06533=1185.164,189.895,-58.342,-177.899,6.626,148.599
C06534=1185.169,189.646,-58.318,-177.902,6.624,148.599
C06535=1185.173,189.397,-58.295,-177.904,6.622,148.599
C06536=1185.178,189.148,-58.272,-177.907,6.620,148.599
C06537=1185.183,188.899,-58.248,-177.909,6.619,148.600
C06538=1185.187,188.651,-58.225,-177.912,6.617,148.600
C06539=1185.191,188.401,-58.202,-177.915,6.615,148.600
C06540=1185.196,188.152,-58.179,-177.917,6.613,148.601
C06541=1185.201,187.903,-58.155,-177.920,6.611,148.601
C06542=1185.205,187.655,-58.133,-177.923,6.609,148.601
C06543=1185.210,187.406,-58.110,-177.926,6.607,148.602
C06544=1185.215,187.157,-58.086,-177.928,6.605,148.602
C06545=1185.220,186.908,-58.063,-177.931,6.603,148.602
C06546=1185.223,186.660,-58.040,-177.934,6.601,148.603
C06547=1185.228,186.411,-58.017,-177.936,6.599,148.603
C06548=1185.233,186.162,-57.993,-177.939,6.598,148.603
C06549=1185.238,185.913,-57.970,-177.942,6.596,148.604
C06550=1185.242,185.664,-57.948,-177.944,6.594,148.604
C06551=1185.247,185.415,-57.924,-177.946,6.592,148.604
C06552=1185.252,185.166,-57.901,-177.949,6.590,148.605
C06553=1185.256,184.897,-57.877,-177.952,6.588,148.605
C06554=1185.261,184.627,-57.851,-177.955,6.586,148.605
C06555=1185.267,184.357,-57.826,-177.958,6.584,148.606
C06556=1185.271,184.088,-57.802,-177.961,6.582,148.606
C06557=1185.276,183.839,-57.779,-177.964,6.580,148.607
C06558=1185.281,183.591,-57.756,-177.966,6.578,148.607
C06559=1185.286,183.341,-57.734,-177.969,6.576,148.607
C06560=1185.290,183.092,-57.710,-177.972,6.574,148.607
C06561=1185.294,182.844,-57.687,-177.974,6.572,148.608
C06562=1185.299,182.594,-57.664,-177.977,6.571,148.608
C06563=1185.305,182.346,-57.642,-177.980,6.569,148.608
C06564=1185.309,182.097,-57.619,-177.982,6.567,148.609
C06565=1185.313,181.848,-57.596,-177.985,6.565,148.609
C06566=1185.318,181.598,-57.574,-177.988,6.564,148.610
C06567=1185.323,181.350,-57.551,-177.990,6.562,148.610
C06568=1185.327,181.101,-57.528,-177.993,6.560,148.610
C06569=1185.331,180.852,-57.505,-177.996,6.558,148.611
C06570=1185.336,180.603,-57.482,-177.998,6.555,148.611
C06571=1185.341,180.355,-57.460,-178.001,6.553,148.611
C06572=1185.346,180.105,-57.437,-178.004,6.552,148.611
C06573=1185.350,179.856,-57.414,-178.006,6.550,148.612
C06574=1185.355,179.607,-57.391,-178.009,6.548,148.612
C06575=1185.360,179.359,-57.369,-178.012,6.546,148.613
C06576=1185.364,179.110,-57.346,-178.014,6.544,148.613
C06577=1185.368,178.861,-57.323,-178.017,6.543,148.613
C06578=1185.374,178.612,-57.301,-178.020,6.541,148.614
C06579=1185.378,178.363,-57.278,-178.022,6.539,148.614
C06580=1185.383,178.114,-57.255,-178.025,6.537,148.614
C06581=1185.387,177.866,-57.233,-178.028,6.536,148.615
C06582=1185.392,177.616,-57.210,-178.030,6.534,148.615
C06583=1185.396,177.367,-57.187,-178.033,6.532,148.615
C06584=1185.401,177.118,-57.165,-178.036,6.530,148.616
C06585=1185.406,176.869,-57.142,-178.038,6.528,148.616
C06586=1185.410,176.620,-57.120,-178.041,6.527,148.616
C06587=1185.415,176.372,-57.097,-178.044,6.525,148.617
C06588=1185.420,176.122,-57.075,-178.046,6.523,148.617
C06589=1185.424,175.873,-57.052,-178.049,6.521,148.617
C06590=1185.429,175.625,-57.030,-178.051,6.519,148.618
C06591=1185.434,175.375,-57.008,-178.054,6.517,148.618
C06592=1185.438,175.126,-56.985,-178.057,6.516,148.618
C06593=1185.443,174.878,-56.963,-178.059,6.514,148.619
C06594=1185.448,174.629,-56.940,-178.062,6.512,148.619
C06595=1185.452,174.379,-56.918,-178.065,6.510,148.620
C06596=1185.457,174.131,-56.896,-178.067,6.508,148.620
C06597=1185.462,173.882,-56.873,-178.070,6.507,148.620
C06598=1185.467,173.633,-56.851,-178.073,6.505,148.621
C06599=1185.471,173.384,-56.829,-178.075,6.503,148.621
C06600=1185.476,173.135,-56.806,-178.078,6.501,148.621
C06601=1185.480,172.886,-56.784,-178.081,6.500,148.622
C06602=1185.485,172.637,-56.762,-178.083,6.498,148.622
C06603=1185.490,172.388,-56.739,-178.086,6.496,148.622
C06604=1185.494,172.139,-56.717,-178.089,6.494,148.623
C06605=1185.499,171.890,-56.695,-178.091,6.492,148.623
C06606=1185.503,171.642,-56.672,-178.094,6.491,148.624
C06607=1185.508,171.392,-56.650,-178.097,6.489,148.624
C06608=1185.513,171.143,-56.628,-178.100,6.487,148.624
C06609=1185.517,170.894,-56.606,-178.102,6.485,148.625
C06610=1185.523,170.645,-56.584,-178.105,6.484,148.625
C06611=1185.527,170.396,-56.561,-178.108,6.482,148.625
C06612=1185.532,170.148,-56.539,-178.110,6.480,148.626
C06613=1185.536,169.898,-56.517,-178.113,6.478,148.626
C06614=1185.541,169.650,-56.496,-178.116,6.476,148.626
C06615=1185.546,169.400,-56.473,-178.118,6.475,148.627
C06616=1185.551,169.151,-56.451,-178.121,6.473,148.627
C06617=1185.555,168.903,-56.429,-178.124,6.471,148.628
C06618=1185.559,168.654,-56.407,-178.126,6.469,148.628
C06619=1185.565,168.404,-56.384,-178.129,6.468,148.628
C06620=1185.569,168.156,-56.363,-178.132,6.466,148.629
C06621=1185.574,167.906,-56.340,-178.134,6.464,148.629
C06622=1185.579,167.658,-56.319,-178.137,6.462,148.629
C06623=1185.583,167.409,-56.297,-178.139,6.461,148.630
C06624=1185.588,167.160,-56.275,-178.142,6.459,148.630
C06625=1185.593,166.910,-56.252,-178.144,6.458,148.630
C06626=1185.598,166.662,-56.231,-178.147,6.456,148.631
C06627=1185.602,166.412,-56.209,-178.150,6.454,148.631
C06628=1185.607,166.164,-56.187,-178.152,6.452,148.632
C06629=1185.611,165.914,-56.165,-178.155,6.451,148.632
C06630=1185.616,165.666,-56.143,-178.158,6.449,148.632
C06631=1185.620,165.416,-56.121,-178.161,6.447,148.633
C06632=1185.625,165.168,-56.100,-178.164,6.446,148.633
C06633=1185.629,164.918,-56.077,-178.166,6.444,148.634
C06634=1185.634,164.670,-56.056,-178.169,6.442,148.634
C06635=1185.639,164.421,-56.034,-178.172,6.440,148.634
C06636=1185.644,164.171,-56.011,-178.174,6.438,148.635
C06637=1185.649,163.923,-55.990,-178.177,6.437,148.635
C06638=1185.653,163.673,-55.968,-178.180,6.435,148.636
C06639=1185.658,163.425,-55.946,-178.182,6.433,148.636
C06640=1185.662,163.175,-55.924,-178.185,6.432,148.636
C06641=1185.667,162.927,-55.902,-178.187,6.430,148.637
C06642=1185.672,162.678,-55.881,-178.190,6.429,148.637
C06643=1185.677,162.428,-55.859,-178.193,6.427,148.637
C06644=1185.681,162.180,-55.838,-178.195,6.425,148.638
C06645=1185.686,161.930,-55.816,-178.198,6.423,148.638
C06646=1185.691,161.682,-55.794,-178.201,6.422,148.638
C06647=1185.695,161.433,-55.772,-178.203,6.420,148.639
C06648=1185.700,161.184,-55.750,-178.206,6.418,148.639
C06649=1185.705,160.934,-55.729,-178.209,6.416,148.640
C06650=1185.710,160.686,-55.708,-178.212,6.415,148.640
C06651=1185.714,160.436,-55.685,-178.215,6.413,148.641
C06652=1185.718,160.188,-55.664,-178.217,6.412,148.641
C06653=1185.723,159.939,-55.643,-178.219,6.410,148.641
C06654=1185.728,159.689,-55.621,-178.222,6.409,148.642
C06655=1185.732,159.441,-55.600,-178.225,6.407,148.642
C06656=1185.737,159.191,-55.578,-178.227,6.405,148.642
C06657=1185.743,158.923,-55.555,-178.230,6.403,148.643
C06658=1185.748,158.654,-55.532,-178.233,6.401,148.643
C06659=1185.753,158.384,-55.509,-178.236,6.400,148.644
C06660=1185.757,158.116,-55.485,-178.239,6.397,148.644
C06661=1185.762,157.866,-55.464,-178.241,6.396,148.645
C06662=1185.767,157.617,-55.442,-178.244,6.395,148.645
C06663=1185.772,157.369,-55.420,-178.247,6.393,148.645
C06664=1185.777,157.119,-55.399,-178.249,6.391,148.646
C06665=1185.781,156.870,-55.377,-178.252,6.389,148.646
C06666=1185.786,156.621,-55.357,-178.255,6.388,148.646
C06667=1185.791,156.372,-55.335,-178.258,6.386,148.647
C06668=1185.795,156.123,-55.313,-178.261,6.384,148.647
C06669=1185.800,155.874,-55.292,-178.263,6.383,148.648
C06670=1185.805,155.625,-55.271,-178.265,6.382,148.648
C06671=1185.809,155.376,-55.250,-178.268,6.380,148.649
C06672=1185.814,155.127,-55.228,-178.271,6.378,148.649
C06673=1185.819,154.878,-55.207,-178.273,6.376,148.649
C06674=1185.824,154.629,-55.186,-178.276,6.375,148.650
C06675=1185.829,154.380,-55.165,-178.279,6.373,148.650
C06676=1185.832,154.131,-55.143,-178.282,6.371,148.651
C06677=1185.837,153.881,-55.122,-178.284,6.370,148.651
C06678=1185.842,153.633,-55.100,-178.287,6.369,148.651
C06679=1185.848,153.384,-55.079,-178.289,6.367,148.652
C06680=1185.851,153.135,-55.058,-178.292,6.365,148.652
C06681=1185.856,152.885,-55.037,-178.295,6.363,148.653
C06682=1185.861,152.637,-55.015,-178.297,6.362,148.653
C06683=1185.866,152.387,-54.994,-178.300,6.360,148.653
C06684=1185.871,152.138,-54.974,-178.302,6.359,148.654
C06685=1185.875,151.889,-54.952,-178.305,6.357,148.654
C06686=1185.880,151.640,-54.931,-178.308,6.356,148.655
C06687=1185.884,151.392,-54.910,-178.311,6.354,148.655
C06688=1185.889,151.142,-54.889,-178.313,6.352,148.655
C06689=1185.895,150.893,-54.868,-178.316,6.350,148.656
C06690=1185.899,150.645,-54.847,-178.318,6.349,148.656
C06691=1185.903,150.395,-54.826,-178.321,6.348,148.657
C06692=1185.908,150.145,-54.805,-178.324,6.346,148.657
C06693=1185.913,149.897,-54.784,-178.327,6.345,148.658
C06694=1185.918,149.648,-54.763,-178.329,6.343,148.658
C06695=1185.923,149.399,-54.742,-178.332,6.341,148.658
C06696=1185.927,149.150,-54.721,-178.334,6.340,148.659
C06697=1185.932,148.900,-54.699,-178.337,6.338,148.659
C06698=1185.937,148.651,-54.678,-178.340,6.337,148.659
C06699=1185.941,148.402,-54.658,-178.343,6.335,148.660
C06700=1185.946,148.153,-54.636,-178.346,6.333,148.660
C06701=1185.951,147.905,-54.616,-178.348,6.332,148.661
C06702=1185.956,147.655,-54.595,-178.350,6.331,148.661
C06703=1185.960,147.406,-54.574,-178.353,6.329,148.662
C06704=1185.965,147.157,-54.553,-178.356,6.327,148.662
C06705=1185.970,146.908,-54.531,-178.358,6.325,148.662
C06706=1185.974,146.659,-54.511,-178.362,6.324,148.663
C06707=1185.979,146.410,-54.490,-178.364,6.323,148.663
C06708=1185.984,146.161,-54.470,-178.366,6.321,148.664
C06709=1185.989,145.911,-54.449,-178.369,6.319,148.664
C06710=1185.993,145.662,-54.428,-178.372,6.318,148.665
C06711=1185.998,145.413,-54.407,-178.374,6.316,148.665
C06712=1186.003,145.165,-54.386,-178.378,6.314,148.665
C06713=1186.008,144.916,-54.365,-178.380,6.314,148.666
C06714=1186.012,144.667,-54.345,-178.382,6.312,148.666
C06715=1186.017,144.417,-54.324,-178.385,6.310,148.667
C06716=1186.022,144.168,-54.304,-178.388,6.308,148.667
C06717=1186.026,143.918,-54.282,-178.391,6.307,148.668
C06718=1186.031,143.669,-54.262,-178.393,6.306,148.668
C06719=1186.036,143.420,-54.241,-178.396,6.304,148.668
C06720=1186.040,143.171,-54.221,-178.398,6.302,148.669
C06721=1186.046,142.922,-54.200,-178.401,6.301,148.669
C06722=1186.050,142.673,-54.179,-178.403,6.300,148.670
C06723=1186.055,142.424,-54.159,-178.406,6.298,148.670
C06724=1186.060,142.175,-54.138,-178.409,6.296,148.671
C06725=1186.064,141.926,-54.118,-178.412,6.295,148.671
C06726=1186.069,141.677,-54.097,-178.414,6.293,148.671
C06727=1186.074,141.428,-54.076,-178.417,6.292,148.672
C06728=1186.078,141.179,-54.056,-178.420,6.291,148.672
C06729=1186.083,140.929,-54.035,-178.422,6.289,148.673
C06730=1186.088,140.680,-54.015,-178.425,6.287,148.673
C06731=1186.093,140.431,-53.994,-178.427,6.286,148.674
C06732=1186.097,140.182,-53.973,-178.430,6.284,148.674
C06733=1186.102,139.933,-53.953,-178.433,6.283,148.675
C06734=1186.107,139.683,-53.933,-178.436,6.281,148.675
C06735=1186.112,139.435,-53.912,-178.439,6.279,148.675
C06736=1186.116,139.186,-53.892,-178.441,6.279,148.676
C06737=1186.121,138.936,-53.871,-178.443,6.277,148.676
C06738=1186.126,138.687,-53.850,-178.447,6.275,148.677
C06739=1186.130,138.438,-53.830,-178.449,6.274,148.677
C06740=1186.135,138.189,-53.809,-178.451,6.273,148.677
C06741=1186.140,137.940,-53.789,-178.454,6.271,148.678
C06742=1186.145,137.691,-53.769,-178.457,6.269,148.678
C06743=1186.150,137.442,-53.749,-178.460,6.268,148.679
C06744=1186.155,137.193,-53.728,-178.462,6.267,148.679
C06745=1186.160,136.944,-53.708,-178.465,6.265,148.680
C06746=1186.164,136.695,-53.688,-178.467,6.263,148.680
C06747=1186.168,136.446,-53.668,-178.471,6.262,148.681
C06748=1186.174,136.196,-53.647,-178.473,6.261,148.681
C06749=1186.178,135.947,-53.627,-178.475,6.259,148.681
C06750=1186.183,135.698,-53.607,-178.478,6.257,148.682
C06751=1186.187,135.449,-53.586,-178.481,6.256,148.682
C06752=1186.192,135.200,-53.565,-178.483,6.255,148.683
C06753=1186.198,134.951,-53.546,-178.486,6.253,148.683
C06754=1186.202,134.702,-53.526,-178.489,6.252,148.684
C06755=1186.207,134.453,-53.505,-178.491,6.251,148.684
C06756=1186.212,134.203,-53.485,-178.494,6.249,148.685
C06757=1186.217,133.954,-53.465,-178.497,6.247,148.685
C06758=1186.221,133.704,-53.445,-178.499,6.246,148.685
C06759=1186.226,133.456,-53.425,-178.502,6.245,148.686
C06760=1186.230,133.207,-53.404,-178.505,6.243,148.686
C06761=1186.236,132.938,-53.383,-178.507,6.242,148.687
C06762=1186.240,132.670,-53.361,-178.510,6.240,148.687
C06763=1186.246,132.401,-53.339,-178.513,6.238,148.688
C06764=1186.251,132.132,-53.318,-178.516,6.237,148.688
C06765=1186.255,131.883,-53.298,-178.519,6.235,148.689
C06766=1186.261,131.634,-53.278,-178.521,6.234,148.689
C06767=1186.266,131.385,-53.257,-178.524,6.233,148.690
C06768=1186.271,131.135,-53.238,-178.527,6.231,148.690
C06769=1186.275,130.886,-53.217,-178.529,6.230,148.691
C06770=1186.280,130.637,-53.198,-178.532,6.228,148.691
C06771=1186.285,130.389,-53.178,-178.535,6.227,148.691
C06772=1186.290,130.139,-53.158,-178.537,6.226,148.692
C06773=1186.294,129.890,-53.138,-178.540,6.224,148.692
C06774=1186.299,129.641,-53.118,-178.543,6.223,148.693
C06775=1186.303,129.392,-53.098,-178.545,6.221,148.693
C06776=1186.309,129.143,-53.078,-178.547,6.220,148.694
C06777=1186.313,128.894,-53.058,-178.551,6.219,148.694
C06778=1186.318,128.644,-53.038,-178.553,6.217,148.695
C06779=1186.323,128.395,-53.017,-178.555,6.216,148.695
C06780=1186.328,128.145,-52.998,-178.559,6.214,148.696
C06781=1186.333,127.896,-52.978,-178.561,6.213,148.696
C06782=1186.337,127.648,-52.958,-178.563,6.212,148.696
C06783=1186.342,127.398,-52.938,-178.566,6.210,148.697
C06784=1186.347,127.148,-52.919,-178.569,6.209,148.697
C06785=1186.352,126.900,-52.899,-178.571,6.208,148.698
C06786=1186.357,126.651,-52.879,-178.574,6.206,148.698
C06787=1186.361,126.401,-52.860,-178.577,6.204,148.699
C06788=1186.365,126.152,-52.840,-178.579,6.204,148.699
C06789=1186.371,125.904,-52.820,-178.582,6.202,148.700
C06790=1186.375,125.654,-52.801,-178.585,6.200,148.700
C06791=1186.380,125.405,-52.780,-178.588,6.199,148.701
C06792=1186.385,125.156,-52.761,-178.590,6.198,148.701
C06793=1186.390,124.907,-52.741,-178.593,6.196,148.702
C06794=1186.394,124.658,-52.721,-178.596,6.195,148.702
C06795=1186.399,124.408,-52.701,-178.598,6.194,148.703
C06796=1186.404,124.159,-52.682,-178.601,6.192,148.703
C06797=1186.409,123.910,-52.662,-178.604,6.190,148.703
C06798=1186.414,123.660,-52.643,-178.606,6.190,148.704
C06799=1186.419,123.412,-52.623,-178.609,6.188,148.704
C06800=1186.423,123.163,-52.604,-178.611,6.187,148.705
C06801=1186.428,122.913,-52.584,-178.614,6.186,148.705
C06802=1186.433,122.664,-52.565,-178.617,6.184,148.706
C06803=1186.438,122.415,-52.545,-178.619,6.183,148.706
C06804=1186.442,122.166,-52.525,-178.622,6.181,148.707
C06805=1186.447,121.917,-52.505,-178.625,6.180,148.707
C06806=1186.452,121.667,-52.486,-178.627,6.179,148.708
C06807=1186.456,121.418,-52.467,-178.630,6.177,148.708
C06808=1186.462,121.169,-52.447,-178.633,6.176,148.709
C06809=1186.466,120.919,-52.428,-178.635,6.175,148.709
C06810=1186.471,120.670,-52.408,-178.638,6.173,148.709
C06811=1186.476,120.421,-52.389,-178.641,6.172,148.710
C06812=1186.481,120.171,-52.369,-178.643,6.171,148.710
C06813=1186.485,119.924,-52.350,-178.646,6.169,148.711
C06814=1186.490,119.674,-52.330,-178.648,6.168,148.712
C06815=1186.495,119.424,-52.310,-178.651,6.167,148.712
C06816=1186.500,119.176,-52.291,-178.654,6.165,148.712
C06817=1186.504,118.926,-52.272,-178.656,6.164,148.713
C06818=1186.510,118.677,-52.253,-178.659,6.163,148.713
C06819=1186.514,118.428,-52.233,-178.662,6.161,148.714
C06820=1186.519,118.178,-52.214,-178.664,6.160,148.714
C06821=1186.524,117.930,-52.195,-178.667,6.158,148.715
C06822=1186.528,117.680,-52.175,-178.670,6.157,148.715
C06823=1186.534,117.431,-52.156,-178.672,6.156,148.716
C06824=1186.539,117.182,-52.136,-178.675,6.154,148.716
C06825=1186.543,116.932,-52.117,-178.677,6.153,148.717
C06826=1186.548,116.683,-52.099,-178.680,6.152,148.717
C06827=1186.553,116.433,-52.079,-178.683,6.150,148.718
C06828=1186.558,116.185,-52.060,-178.685,6.149,148.718
C06829=1186.562,115.935,-52.041,-178.688,6.148,148.719
C06830=1186.568,115.686,-52.021,-178.691,6.147,148.719
C06831=1186.572,115.437,-52.002,-178.693,6.145,148.720
C06832=1186.577,115.188,-51.983,-178.696,6.144,148.720
C06833=1186.582,114.939,-51.963,-178.699,6.143,148.721
C06834=1186.586,114.690,-51.945,-178.701,6.141,148.721
C06835=1186.591,114.440,-51.926,-178.704,6.141,148.722
C06836=1186.597,114.191,-51.906,-178.707,6.139,148.722
C06837=1186.601,113.942,-51.887,-178.710,6.138,148.723
C06838=1186.606,113.693,-51.868,-178.712,6.137,148.723
C06839=1186.611,113.443,-51.848,-178.715,6.135,148.723
C06840=1186.616,113.194,-51.830,-178.717,6.134,148.724
C06841=1186.620,112.945,-51.811,-178.720,6.133,148.724
C06842=1186.625,112.696,-51.792,-178.723,6.131,148.725
C06843=1186.630,112.447,-51.772,-178.725,6.130,148.726
C06844=1186.635,112.198,-51.753,-178.728,6.129,148.726
C06845=1186.639,111.948,-51.735,-178.730,6.128,148.726
C06846=1186.645,111.699,-51.715,-178.733,6.126,148.727
C06847=1186.649,111.450,-51.696,-178.735,6.125,148.727
C06848=1186.654,111.200,-51.678,-178.739,6.124,148.728
C06849=1186.658,110.951,-51.659,-178.741,6.122,148.728
C06850=1186.664,110.702,-51.639,-178.743,6.121,148.729
C06851=1186.669,110.452,-51.620,-178.747,6.120,148.729
C06852=1186.673,110.203,-51.602,-178.749,6.119,148.730
C06853=1186.678,109.954,-51.582,-178.751,6.117,148.730
C06854=1186.683,109.705,-51.563,-178.754,6.117,148.731
C06855=1186.688,109.456,-51.545,-178.757,6.115,148.731
C06856=1186.692,109.206,-51.526,-178.760,6.114,148.732
C06857=1186.698,108.957,-51.507,-178.762,6.113,148.732
C06858=1186.702,108.708,-51.488,-178.765,6.111,148.733
C06859=1186.707,108.459,-51.469,-178.767,6.110,148.733
C06860=1186.712,108.209,-51.451,-178.770,6.109,148.734
C06861=1186.716,107.960,-51.432,-178.772,6.108,148.734
C06862=1186.722,107.711,-51.413,-178.775,6.106,148.735
C06863=1186.726,107.462,-51.394,-178.778,6.104,148.735
C06864=1186.731,107.213,-51.375,-178.781,6.104,148.736
C06865=1186.736,106.945,-51.356,-178.783,6.102,148.736
C06866=1186.742,106.675,-51.335,-178.787,6.101,148.737
C06867=1186.747,106.407,-51.314,-178.789,6.100,148.737
C06868=1186.752,106.139,-51.295,-178.792,6.099,148.738
C06869=1186.757,105.889,-51.275,-178.795,6.097,148.738
C06870=1186.762,105.640,-51.257,-178.797,6.096,148.739
C06871=1186.766,105.391,-51.238,-178.800,6.094,148.739
C06872=1186.772,105.142,-51.220,-178.803,6.094,148.740
C06873=1186.776,104.893,-51.201,-178.805,6.092,148.740
C06874=1186.781,104.643,-51.182,-178.807,6.091,148.741
C06875=1186.786,104.394,-51.163,-178.811,6.090,148.742
C06876=1186.791,104.145,-51.145,-178.813,6.089,148.742
C06877=1186.796,103.895,-51.126,-178.816,6.088,148.743
C06878=1186.800,103.646,-51.108,-178.818,6.087,148.743
C06879=1186.805,103.397,-51.090,-178.821,6.085,148.743
C06880=1186.810,103.148,-51.070,-178.823,6.084,148.744
C06881=1186.815,102.898,-51.052,-178.826,6.083,148.744
C06882=1186.820,102.649,-51.034,-178.829,6.081,148.745
C06883=1186.825,102.400,-51.015,-178.831,6.080,148.746
C06884=1186.830,102.150,-50.997,-178.835,6.079,148.746
C06885=1186.834,101.902,-50.978,-178.837,6.078,148.747
C06886=1186.840,101.652,-50.959,-178.840,6.076,148.747
C06887=1186.844,101.403,-50.941,-178.842,6.076,148.748
C06888=1186.849,101.154,-50.922,-178.845,6.074,148.748
C06889=1186.854,100.905,-50.904,-178.847,6.073,148.749
C06890=1186.859,100.655,-50.885,-178.850,6.072,148.749
C06891=1186.864,100.405,-50.867,-178.853,6.071,148.750
C06892=1186.868,100.157,-50.849,-178.856,6.069,148.750
C06893=1186.873,99.908,-50.831,-178.858,6.068,148.751
C06894=1186.878,99.658,-50.812,-178.861,6.067,148.751
C06895=1186.883,99.408,-50.794,-178.863,6.066,148.752
C06896=1186.888,99.160,-50.775,-178.866,6.065,148.752
C06897=1186.893,98.911,-50.757,-178.868,6.064,148.753
C06898=1186.898,98.660,-50.738,-178.871,6.063,148.753
C06899=1186.903,98.411,-50.720,-178.874,6.062,148.754
C06900=1186.907,98.163,-50.701,-178.876,6.060,148.754
C06901=1186.912,97.914,-50.683,-178.879,6.059,148.755
C06902=1186.916,97.664,-50.665,-178.882,6.058,148.755
C06903=1186.922,97.414,-50.647,-178.884,6.057,148.756
C06904=1186.927,97.165,-50.629,-178.887,6.055,148.756
C06905=1186.932,96.916,-50.611,-178.890,6.055,148.757
C06906=1186.936,96.667,-50.592,-178.892,6.053,148.757
C06907=1186.941,96.417,-50.574,-178.895,6.052,148.758
C06908=1186.946,96.168,-50.556,-178.898,6.051,148.758
C06909=1186.951,95.919,-50.538,-178.900,6.050,148.759
C06910=1186.956,95.670,-50.519,-178.903,6.048,148.759
C06911=1186.961,95.420,-50.501,-178.905,6.048,148.760
C06912=1186.965,95.171,-50.483,-178.908,6.047,148.761
C06913=1186.970,94.921,-50.465,-178.910,6.045,148.761
C06914=1186.975,94.672,-50.447,-178.913,6.045,148.762
C06915=1186.980,94.423,-50.429,-178.916,6.043,148.762
C06916=1186.985,94.174,-50.411,-178.918,6.042,148.763
C06917=1186.989,93.924,-50.392,-178.921,6.041,148.763
C06918=1186.994,93.675,-50.374,-178.924,6.040,148.764
C06919=1187.000,93.426,-50.355,-178.926,6.038,148.764
C06920=1187.005,93.177,-50.337,-178.929,6.037,148.765
C06921=1187.010,92.928,-50.319,-178.932,6.036,148.765
C06922=1187.014,92.678,-50.301,-178.934,6.035,148.766
C06923=1187.020,92.429,-50.284,-178.937,6.034,148.766
C06924=1187.024,92.179,-50.266,-178.939,6.033,148.767
C06925=1187.029,91.930,-50.248,-178.942,6.032,148.767
C06926=1187.034,91.680,-50.230,-178.945,6.031,148.768
C06927=1187.039,91.431,-50.212,-178.947,6.030,148.768
C06928=1187.044,91.182,-50.194,-178.950,6.028,148.769
C06929=1187.049,90.933,-50.176,-178.953,6.028,148.769
C06930=1187.053,90.684,-50.158,-178.955,6.026,148.770
C06931=1187.058,90.434,-50.140,-178.958,6.025,148.771
C06932=1187.063,90.185,-50.121,-178.961,6.024,148.771
C06933=1187.068,89.935,-50.103,-178.963,6.023,148.772
C06934=1187.072,89.686,-50.085,-178.966,6.021,148.772
C06935=1187.078,89.436,-50.068,-178.969,6.021,148.773
C06936=1187.083,89.187,-50.050,-178.971,6.020,148.773
C06937=1187.088,88.938,-50.032,-178.974,6.019,148.774
C06938=1187.092,88.689,-50.014,-178.976,6.018,148.774
C06939=1187.097,88.440,-49.996,-178.979,6.016,148.775
C06940=1187.102,88.191,-49.979,-178.981,6.015,148.775
C06941=1187.107,87.941,-49.962,-178.984,6.014,148.776
C06942=1187.112,87.692,-49.944,-178.987,6.013,148.776
C06943=1187.117,87.443,-49.926,-178.989,6.012,148.777
C06944=1187.121,87.194,-49.908,-178.992,6.011,148.777
C06945=1187.126,86.944,-49.890,-178.994,6.010,148.778
C06946=1187.132,86.695,-49.872,-178.997,6.009,148.778
C06947=1187.136,86.445,-49.854,-179.000,6.008,148.779
C06948=1187.141,86.196,-49.836,-179.003,6.006,148.779
C06949=1187.146,85.946,-49.818,-179.005,6.005,148.780
C06950=1187.150,85.697,-49.801,-179.008,6.005,148.781
C06951=1187.155,85.448,-49.783,-179.010,6.003,148.781
C06952=1187.160,85.199,-49.765,-179.013,6.003,148.782
C06953=1187.165,84.949,-49.748,-179.016,6.001,148.782
C06954=1187.170,84.700,-49.730,-179.018,6.000,148.783
C06955=1187.175,84.450,-49.712,-179.020,5.999,148.783
C06956=1187.180,84.201,-49.696,-179.024,5.998,148.784
C06957=1187.184,83.952,-49.678,-179.026,5.997,148.784
C06958=1187.189,83.703,-49.660,-179.029,5.996,148.785
C06959=1187.195,83.453,-49.642,-179.031,5.995,148.785
C06960=1187.200,83.204,-49.624,-179.034,5.994,148.786
C06961=1187.204,82.954,-49.606,-179.036,5.993,148.786
C06962=1187.209,82.705,-49.590,-179.039,5.992,148.787
C06963=1187.214,82.456,-49.572,-179.042,5.990,148.787
C06964=1187.220,82.207,-49.555,-179.044,5.990,148.788
C06965=1187.225,81.957,-49.537,-179.047,5.989,148.789
C06966=1187.229,81.708,-49.520,-179.050,5.988,148.789
C06967=1187.234,81.459,-49.502,-179.052,5.987,148.790
C06968=1187.239,81.210,-49.484,-179.055,5.985,148.790
C06969=1187.244,80.941,-49.466,-179.058,5.985,148.791
C06970=1187.250,80.672,-49.447,-179.060,5.983,148.791
C06971=1187.254,80.404,-49.428,-179.063,5.983,148.792
C06972=1187.260,80.136,-49.410,-179.066,5.981,148.793
C06973=1187.265,79.887,-49.392,-179.068,5.980,148.793
C06974=1187.270,79.637,-49.374,-179.072,5.979,148.794
C06975=1187.274,79.388,-49.357,-179.074,5.978,148.794
C06976=1187.279,79.138,-49.340,-179.076,5.977,148.795
C06977=1187.284,78.889,-49.322,-179.080,5.976,148.795
C06978=1187.289,78.639,-49.305,-179.082,5.975,148.796
C06979=1187.294,78.390,-49.287,-179.085,5.974,148.797
C06980=1187.299,78.141,-49.270,-179.087,5.973,148.797
C06981=1187.304,77.892,-49.254,-179.090,5.972,148.798
C06982=1187.309,77.643,-49.236,-179.092,5.971,148.798
C06983=1187.314,77.393,-49.218,-179.095,5.970,148.799
C06984=1187.318,77.144,-49.201,-179.097,5.969,148.799
C06985=1187.324,76.894,-49.184,-179.100,5.968,148.800
C06986=1187.329,76.644,-49.166,-179.102,5.967,148.800
C06987=1187.333,76.395,-49.149,-179.105,5.966,148.801
C06988=1187.338,76.146,-49.132,-179.108,5.965,148.801
C06989=1187.343,75.897,-49.116,-179.110,5.964,148.802
C06990=1187.348,75.648,-49.098,-179.114,5.963,148.803
C06991=1187.353,75.398,-49.080,-179.116,5.962,148.803
C06992=1187.358,75.148,-49.064,-179.118,5.961,148.804
C06993=1187.363,74.899,-49.046,-179.121,5.960,148.804
C06994=1187.367,74.650,-49.029,-179.124,5.959,148.805
C06995=1187.373,74.401,-49.012,-179.126,5.958,148.805
C06996=1187.378,74.151,-48.994,-179.129,5.957,148.806
C06997=1187.383,73.902,-48.977,-179.131,5.956,148.806
C06998=1187.388,73.652,-48.960,-179.134,5.955,148.807
C06999=1187.392,73.403,-48.943,-179.137,5.954,148.807
C07000=1187.397,73.154,-48.926,-179.139,5.953,148.808
C07001=1187.402,72.905,-48.909,-179.142,5.953,148.809
C07002=1187.407,72.655,-48.892,-179.145,5.951,148.809
C07003=1187.412,72.405,-48.875,-179.147,5.950,148.810
C07004=1187.417,72.156,-48.857,-179.149,5.949,148.810
C07005=1187.421,71.907,-48.841,-179.153,5.948,148.811
C07006=1187.427,71.658,-48.824,-179.155,5.947,148.811
C07007=1187.432,71.408,-48.807,-179.157,5.947,148.812
C07008=1187.437,71.158,-48.790,-179.160,5.945,148.812
C07009=1187.441,70.909,-48.773,-179.163,5.944,148.813
C07010=1187.447,70.660,-48.756,-179.165,5.944,148.814
C07011=1187.451,70.411,-48.739,-179.168,5.942,148.814
C07012=1187.457,70.161,-48.722,-179.171,5.942,148.815
C07013=1187.461,69.912,-48.705,-179.173,5.941,148.815
C07014=1187.467,69.663,-48.688,-179.176,5.939,148.816
C07015=1187.471,69.413,-48.671,-179.178,5.939,148.816
C07016=1187.476,69.164,-48.655,-179.181,5.938,148.817
C07017=1187.481,68.914,-48.637,-179.184,5.937,148.818
C07018=1187.486,68.665,-48.621,-179.186,5.936,148.818
C07019=1187.491,68.416,-48.603,-179.189,5.935,148.819
C07020=1187.495,68.166,-48.586,-179.191,5.934,148.819
C07021=1187.501,67.917,-48.569,-179.194,5.933,148.820
C07022=1187.506,67.668,-48.553,-179.196,5.932,148.820
C07023=1187.510,67.418,-48.536,-179.199,5.932,148.821
C07024=1187.515,67.169,-48.519,-179.202,5.930,148.822
C07025=1187.521,66.920,-48.503,-179.204,5.929,148.822
C07026=1187.525,66.670,-48.486,-179.207,5.929,148.823
C07027=1187.530,66.420,-48.469,-179.210,5.927,148.823
C07028=1187.535,66.171,-48.452,-179.212,5.926,148.824
C07029=1187.540,65.922,-48.436,-179.215,5.926,148.824
C07030=1187.545,65.672,-48.418,-179.218,5.924,148.825
C07031=1187.549,65.423,-48.402,-179.220,5.924,148.825
C07032=1187.555,65.174,-48.386,-179.222,5.923,148.826
C07033=1187.560,64.924,-48.368,-179.225,5.922,148.827
C07034=1187.565,64.674,-48.352,-179.228,5.921,148.827
C07035=1187.570,64.425,-48.336,-179.230,5.920,148.828
C07036=1187.575,64.176,-48.319,-179.233,5.920,148.828
C07037=1187.579,63.926,-48.302,-179.236,5.918,148.829
C07038=1187.584,63.677,-48.286,-179.238,5.917,148.829
C07039=1187.590,63.428,-48.268,-179.241,5.916,148.830
C07040=1187.594,63.178,-48.252,-179.243,5.916,148.831
C07041=1187.599,62.929,-48.236,-179.246,5.915,148.831
C07042=1187.604,62.680,-48.219,-179.249,5.914,148.832
C07043=1187.609,62.429,-48.202,-179.251,5.913,148.832
C07044=1187.614,62.181,-48.186,-179.253,5.912,148.833
C07045=1187.619,61.931,-48.169,-179.257,5.911,148.833
C07046=1187.624,61.682,-48.153,-179.259,5.910,148.834
C07047=1187.629,61.433,-48.136,-179.261,5.909,148.834
C07048=1187.634,61.183,-48.119,-179.265,5.908,148.835
C07049=1187.639,60.934,-48.103,-179.267,5.907,148.836
C07050=1187.643,60.684,-48.087,-179.269,5.907,148.836
C07051=1187.649,60.435,-48.070,-179.272,5.906,148.837
C07052=1187.654,60.186,-48.053,-179.275,5.904,148.837
C07053=1187.659,59.936,-48.037,-179.277,5.904,148.838
C07054=1187.664,59.687,-48.021,-179.279,5.903,148.838
C07055=1187.668,59.437,-48.004,-179.282,5.902,148.839
C07056=1187.674,59.188,-47.987,-179.285,5.901,148.840
C07057=1187.679,58.938,-47.971,-179.287,5.900,148.840
C07058=1187.684,58.689,-47.955,-179.290,5.900,148.841
C07059=1187.688,58.440,-47.939,-179.292,5.899,148.841
C07060=1187.693,58.190,-47.923,-179.295,5.897,148.842
C07061=1187.698,57.941,-47.906,-179.298,5.897,148.843
C07062=1187.703,57.691,-47.889,-179.300,5.896,148.843
C07063=1187.708,57.442,-47.873,-179.303,5.896,148.844
C07064=1187.713,57.192,-47.857,-179.306,5.894,148.844
C07065=1187.718,56.943,-47.840,-179.308,5.893,148.845
C07066=1187.723,56.693,-47.824,-179.311,5.893,148.845
C07067=1187.728,56.445,-47.808,-179.313,5.892,148.846
C07068=1187.733,56.195,-47.792,-179.316,5.891,148.847
C07069=1187.738,55.946,-47.776,-179.319,5.890,148.847
C07070=1187.742,55.696,-47.759,-179.321,5.889,148.848
C07071=1187.748,55.447,-47.742,-179.324,5.889,148.848
C07072=1187.753,55.197,-47.726,-179.326,5.887,148.849
C07073=1187.759,54.929,-47.709,-179.329,5.886,148.849
C07074=1187.763,54.660,-47.691,-179.332,5.886,148.850
C07075=1187.769,54.392,-47.674,-179.335,5.885,148.851
C07076=1187.774,54.123,-47.657,-179.338,5.884,148.851
C07077=1187.779,53.874,-47.641,-179.340,5.883,148.852
C07078=1187.784,53.625,-47.624,-179.343,5.882,148.853
C07079=1187.789,53.375,-47.608,-179.346,5.881,148.853
C07080=1187.794,53.126,-47.592,-179.348,5.880,148.854
C07081=1187.799,52.876,-47.576,-179.350,5.880,148.854
C07082=1187.804,52.627,-47.560,-179.354,5.879,148.855
C07083=1187.808,52.377,-47.544,-179.356,5.878,148.855
C07084=1187.814,52.128,-47.527,-179.358,5.877,148.856
C07085=1187.819,51.879,-47.512,-179.360,5.876,148.857
C07086=1187.824,51.629,-47.496,-179.363,5.876,148.857
C07087=1187.829,51.380,-47.480,-179.366,5.874,148.858
C07088=1187.834,51.130,-47.464,-179.368,5.874,148.858
C07089=1187.839,50.881,-47.447,-179.371,5.873,148.859
C07090=1187.843,50.631,-47.431,-179.374,5.872,148.860
C07091=1187.849,50.382,-47.415,-179.376,5.872,148.860
C07092=1187.853,50.132,-47.399,-179.379,5.870,148.861
C07093=1187.859,49.883,-47.384,-179.382,5.870,148.861
C07094=1187.864,49.634,-47.367,-179.384,5.869,148.862
C07095=1187.869,49.384,-47.351,-179.387,5.868,148.863
C07096=1187.874,49.135,-47.335,-179.389,5.867,148.863
C07097=1187.878,48.885,-47.319,-179.392,5.866,148.864
C07098=1187.884,48.635,-47.303,-179.395,5.866,148.864
C07099=1187.889,48.387,-47.287,-179.397,5.865,148.865
C07100=1187.893,48.137,-47.272,-179.399,5.864,148.865
C07101=1187.898,47.887,-47.256,-179.402,5.864,148.866
C07102=1187.903,47.638,-47.240,-179.405,5.862,148.867
C07103=1187.908,47.388,-47.224,-179.407,5.861,148.867
C07104=1187.914,47.139,-47.208,-179.410,5.861,148.868
C07105=1187.918,46.889,-47.192,-179.412,5.860,148.868
C07106=1187.923,46.640,-47.176,-179.415,5.860,148.869
C07107=1187.928,46.390,-47.160,-179.418,5.858,148.870
C07108=1187.933,46.141,-47.145,-179.420,5.857,148.870
C07109=1187.938,45.892,-47.129,-179.423,5.857,148.871
C07110=1187.943,45.642,-47.113,-179.425,5.856,148.871
C07111=1187.948,45.393,-47.097,-179.428,5.855,148.872
C07112=1187.954,45.143,-47.082,-179.430,5.855,148.873
C07113=1187.958,44.893,-47.066,-179.433,5.853,148.873
C07114=1187.963,44.645,-47.050,-179.436,5.853,148.874
C07115=1187.968,44.395,-47.035,-179.438,5.852,148.874
C07116=1187.973,44.145,-47.019,-179.440,5.851,148.875
C07117=1187.978,43.896,-47.003,-179.443,5.851,148.875
C07118=1187.984,43.646,-46.987,-179.446,5.850,148.876
C07119=1187.987,43.397,-46.971,-179.448,5.849,148.877
C07120=1187.993,43.148,-46.956,-179.451,5.848,148.877
C07121=1187.998,42.898,-46.940,-179.454,5.848,148.878
C07122=1188.003,42.648,-46.924,-179.456,5.847,148.878
C07123=1188.008,42.399,-46.909,-179.458,5.846,148.879
C07124=1188.013,42.150,-46.894,-179.461,5.846,148.880
C07125=1188.018,41.900,-46.878,-179.464,5.844,148.880
C07126=1188.023,41.650,-46.862,-179.467,5.843,148.881
C07127=1188.027,41.402,-46.846,-179.469,5.843,148.881
C07128=1188.033,41.152,-46.831,-179.471,5.842,148.882
C07129=1188.038,40.902,-46.815,-179.474,5.842,148.883
C07130=1188.043,40.653,-46.799,-179.477,5.841,148.883
C07131=1188.048,40.404,-46.784,-179.479,5.840,148.884
C07132=1188.053,40.154,-46.769,-179.482,5.839,148.884
C07133=1188.058,39.904,-46.753,-179.485,5.838,148.885
C07134=1188.063,39.655,-46.738,-179.487,5.837,148.886
C07135=1188.068,39.406,-46.722,-179.489,5.837,148.886
C07136=1188.073,39.156,-46.707,-179.492,5.836,148.887
C07137=1188.078,38.906,-46.691,-179.494,5.836,148.887
C07138=1188.083,38.657,-46.676,-179.497,5.834,148.888
C07139=1188.088,38.408,-46.660,-179.500,5.834,148.889
C07140=1188.094,38.158,-46.644,-179.502,5.833,148.889
C07141=1188.098,37.909,-46.629,-179.505,5.832,148.890
C07142=1188.103,37.659,-46.613,-179.508,5.832,148.890
C07143=1188.108,37.410,-46.598,-179.510,5.831,148.891
C07144=1188.113,37.161,-46.583,-179.512,5.830,148.892
C07145=1188.118,36.911,-46.567,-179.515,5.830,148.892
C07146=1188.122,36.662,-46.552,-179.518,5.828,148.893
C07147=1188.128,36.412,-46.536,-179.520,5.828,148.893
C07148=1188.133,36.162,-46.521,-179.523,5.827,148.894
C07149=1188.138,35.913,-46.506,-179.526,5.827,148.895
C07150=1188.144,35.664,-46.491,-179.528,5.826,148.895
C07151=1188.148,35.414,-46.476,-179.530,5.825,148.896
C07152=1188.153,35.164,-46.460,-179.533,5.825,148.897
C07153=1188.158,34.915,-46.444,-179.535,5.824,148.897
C07154=1188.163,34.666,-46.429,-179.538,5.823,148.898
C07155=1188.168,34.417,-46.414,-179.541,5.822,148.898
C07156=1188.173,34.167,-46.399,-179.543,5.821,148.899
C07157=1188.178,33.917,-46.384,-179.546,5.821,148.899
C07158=1188.183,33.668,-46.369,-179.549,5.820,148.900
C07159=1188.188,33.418,-46.353,-179.551,5.819,148.901
C07160=1188.193,33.169,-46.338,-179.553,5.819,148.901
C07161=1188.198,32.920,-46.322,-179.556,5.818,148.902
C07162=1188.204,32.670,-46.308,-179.558,5.817,148.902
C07163=1188.208,32.420,-46.292,-179.561,5.816,148.903
C07164=1188.213,32.171,-46.277,-179.564,5.816,148.904
C07165=1188.218,31.921,-46.262,-179.567,5.815,148.904
C07166=1188.224,31.671,-46.247,-179.569,5.814,148.905
C07167=1188.228,31.422,-46.232,-179.571,5.814,148.906
C07168=1188.234,31.173,-46.216,-179.574,5.813,148.906
C07169=1188.238,30.924,-46.201,-179.576,5.812,148.907
C07170=1188.243,30.674,-46.187,-179.579,5.812,148.907
C07171=1188.249,30.425,-46.171,-179.582,5.811,148.908
C07172=1188.253,30.175,-46.156,-179.584,5.810,148.908
C07173=1188.258,29.925,-46.141,-179.587,5.809,148.909
C07174=1188.263,29.676,-46.126,-179.590,5.809,148.910
C07175=1188.268,29.426,-46.110,-179.592,5.808,148.910
C07176=1188.273,29.177,-46.096,-179.594,5.807,148.911
C07177=1188.279,28.908,-46.079,-179.597,5.807,148.912
C07178=1188.284,28.639,-46.063,-179.600,5.806,148.912
C07179=1188.290,28.370,-46.047,-179.603,5.805,148.913
C07180=1188.295,28.102,-46.031,-179.606,5.804,148.914
C07181=1188.300,27.852,-46.016,-179.608,5.804,148.914
C07182=1188.305,27.603,-46.001,-179.610,5.803,148.915
C07183=1188.310,27.353,-45.987,-179.613,5.803,148.915
C07184=1188.315,27.104,-45.971,-179.616,5.802,148.916
C07185=1188.320,26.854,-45.957,-179.618,5.801,148.917
C07186=1188.326,26.605,-45.941,-179.620,5.801,148.917
C07187=1188.330,26.356,-45.926,-179.623,5.800,148.918
C07188=1188.335,26.106,-45.912,-179.625,5.799,148.918
C07189=1188.341,25.857,-45.896,-179.628,5.799,148.919
C07190=1188.346,25.607,-45.882,-179.631,5.798,148.920
C07191=1188.350,25.357,-45.867,-179.634,5.797,148.920
C07192=1188.356,25.107,-45.852,-179.636,5.796,148.921
C07193=1188.360,24.858,-45.837,-179.639,5.796,148.922
C07194=1188.365,24.608,-45.822,-179.641,5.795,148.922
C07195=1188.370,24.359,-45.807,-179.643,5.794,148.923
C07196=1188.375,24.109,-45.793,-179.646,5.794,148.923
C07197=1188.380,23.860,-45.778,-179.649,5.793,148.924
C07198=1188.386,23.610,-45.763,-179.651,5.792,148.924
C07199=1188.390,23.361,-45.748,-179.653,5.792,148.925
C07200=1188.395,23.111,-45.733,-179.656,5.791,148.926
C07201=1188.400,22.862,-45.718,-179.659,5.791,148.927
C07202=1188.406,22.612,-45.704,-179.661,5.790,148.927
C07203=1188.410,22.363,-45.689,-179.664,5.790,148.928
C07204=1188.415,22.113,-45.674,-179.666,5.789,148.928
C07205=1188.421,21.863,-45.659,-179.668,5.788,148.929
C07206=1188.426,21.615,-45.645,-179.671,5.788,148.929
C07207=1188.431,21.365,-45.631,-179.674,5.787,148.930
C07208=1188.436,21.116,-45.616,-179.677,5.786,148.931
C07209=1188.442,20.866,-45.601,-179.679,5.785,148.931
C07210=1188.447,20.616,-45.586,-179.682,5.785,148.932
C07211=1188.451,20.367,-45.571,-179.684,5.784,148.933
C07212=1188.456,20.118,-45.557,-179.687,5.783,148.933
C07213=1188.461,19.868,-45.543,-179.689,5.783,148.934
C07214=1188.466,19.619,-45.527,-179.692,5.782,148.934
C07215=1188.471,19.369,-45.513,-179.694,5.782,148.935
C07216=1188.476,19.119,-45.499,-179.697,5.781,148.936
C07217=1188.481,18.870,-45.484,-179.699,5.780,148.936
C07218=1188.486,18.620,-45.469,-179.702,5.780,148.937
C07219=1188.492,18.370,-45.455,-179.705,5.779,148.938
C07220=1188.496,18.121,-45.440,-179.707,5.778,148.938
C07221=1188.501,17.871,-45.425,-179.709,5.778,148.939
C07222=1188.507,17.622,-45.411,-179.712,5.777,148.939
C07223=1188.512,17.373,-45.397,-179.714,5.777,148.940
C07224=1188.516,17.124,-45.382,-179.717,5.776,148.941
C07225=1188.522,16.874,-45.367,-179.719,5.776,148.941
C07226=1188.527,16.624,-45.353,-179.722,5.775,148.942
C07227=1188.532,16.374,-45.339,-179.724,5.774,148.942
C07228=1188.537,16.125,-45.324,-179.727,5.774,148.943
C07229=1188.542,15.875,-45.309,-179.730,5.773,148.944
C07230=1188.547,15.626,-45.295,-179.732,5.772,148.944
C07231=1188.552,15.377,-45.281,-179.734,5.772,148.945
C07232=1188.557,15.128,-45.266,-179.737,5.771,148.946
C07233=1188.562,14.878,-45.252,-179.740,5.771,148.946
C07234=1188.567,14.628,-45.237,-179.742,5.770,148.947
C07235=1188.572,14.378,-45.223,-179.745,5.770,148.947
C07236=1188.577,14.128,-45.209,-179.747,5.769,148.948
C07237=1188.582,13.879,-45.194,-179.750,5.769,148.949
C07238=1188.588,13.630,-45.180,-179.752,5.768,148.949
C07239=1188.593,13.381,-45.165,-179.755,5.767,148.950
C07240=1188.597,13.131,-45.151,-179.757,5.767,148.951
C07241=1188.602,12.881,-45.137,-179.759,5.766,148.951
C07242=1188.607,12.632,-45.123,-179.762,5.765,148.952
C07243=1188.612,12.382,-45.108,-179.765,5.765,148.952
C07244=1188.618,12.133,-45.094,-179.767,5.764,148.953
C07245=1188.623,11.883,-45.080,-179.770,5.764,148.954
C07246=1188.628,11.633,-45.066,-179.772,5.763,148.954
C07247=1188.633,11.384,-45.052,-179.775,5.763,148.955
C07248=1188.638,11.134,-45.037,-179.778,5.762,148.956
C07249=1188.643,10.885,-45.023,-179.780,5.761,148.956
C07250=1188.648,10.636,-45.008,-179.782,5.761,148.957
C07251=1188.653,10.386,-44.994,-179.785,5.760,148.957
C07252=1188.658,10.136,-44.980,-179.788,5.760,148.958
C07253=1188.663,9.887,-44.966,-179.790,5.759,148.959
C07254=1188.668,9.638,-44.952,-179.792,5.758,148.959
C07255=1188.673,9.388,-44.937,-179.795,5.758,148.960
C07256=1188.678,9.138,-44.923,-179.798,5.757,148.961
C07257=1188.683,8.889,-44.909,-179.800,5.757,148.961
C07258=1188.688,8.639,-44.895,-179.803,5.756,148.962
C07259=1188.694,8.390,-44.881,-179.805,5.756,148.962
C07260=1188.699,8.140,-44.867,-179.807,5.755,148.963
C07261=1188.704,7.890,-44.853,-179.810,5.754,148.964
C07262=1188.709,7.640,-44.838,-179.813,5.754,148.964
C07263=1188.714,7.391,-44.825,-179.815,5.753,148.965
C07264=1188.719,7.141,-44.810,-179.818,5.752,148.965
C07265=1188.724,6.892,-44.797,-179.820,5.752,148.966
C07266=1188.729,6.642,-44.782,-179.823,5.752,148.967
C07267=1188.734,6.393,-44.768,-179.825,5.751,148.968
C07268=1188.739,6.144,-44.754,-179.828,5.750,148.968
C07269=1188.744,5.894,-44.740,-179.830,5.750,148.969
C07270=1188.750,5.645,-44.726,-179.833,5.749,148.969
C07271=1188.755,5.395,-44.712,-179.836,5.749,148.970
C07272=1188.760,5.145,-44.698,-179.838,5.748,148.971
C07273=1188.765,4.895,-44.684,-179.840,5.747,148.971
C07274=1188.770,4.646,-44.671,-179.843,5.747,148.972
C07275=1188.775,4.397,-44.656,-179.846,5.746,148.973
C07276=1188.779,4.147,-44.642,-179.848,5.746,148.973
C07277=1188.785,3.897,-44.629,-179.851,5.745,148.974
C07278=1188.790,3.648,-44.614,-179.853,5.745,148.974
C07279=1188.795,3.398,-44.600,-179.855,5.745,148.975
C07280=1188.800,3.149,-44.587,-179.857,5.744,148.976
C07281=1188.806,2.880,-44.572,-179.860,5.744,148.976
C07282=1188.811,2.610,-44.557,-179.863,5.742,148.977
C07283=1188.816,2.341,-44.542,-179.866,5.742,148.978
C07284=1188.822,2.072,-44.527,-179.869,5.741,148.978
C07285=1188.827,1.823,-44.513,-179.871,5.741,148.979
C07286=1188.832,1.573,-44.499,-179.874,5.740,148.980
C07287=1188.837,1.323,-44.484,-179.876,5.740,148.980
C07288=1188.842,1.074,-44.472,-179.879,5.739,148.981
C07289=1188.847,0.824,-44.458,-179.881,5.739,148.982
C07290=1188.852,0.574,-44.443,-179.883,5.739,148.982
C07291=1188.858,0.325,-44.430,-179.886,5.738,148.983
C07292=1188.862,0.075,-44.416,-179.888,5.738,148.983
C07293=1188.868,-0.174,-44.403,-179.891,5.737,148.984
C07294=1188.873,-0.423,-44.388,-179.894,5.737,148.985
C07295=1188.878,-0.674,-44.375,-179.896,5.736,148.985
C07296=1188.883,-0.922,-44.361,-179.898,5.735,148.986
C07297=1188.888,-1.172,-44.347,-179.901,5.735,148.987
C07298=1188.893,-1.422,-44.334,-179.904,5.734,148.987
C07299=1188.898,-1.671,-44.320,-179.906,5.733,148.988
C07300=1188.903,-1.921,-44.307,-179.909,5.733,148.988
C07301=1188.909,-2.170,-44.293,-179.911,5.733,148.989
